Yaskawa INFORM job: X2_99(90,0)_HARDOX.JBI

/JOB
//NAME X2_99(90,0)_HARDOX
///FOLDERNAME X2
//POS
///NPOS 447,447,443,13,0,0
///TOOL 0
///POSTYPE PULSE
///PULSE
C00000=2000,-99612,-82443,0,53832,0
C00001=-166393,-132062,-92618,58483,55149,81008
C00002=-157482,-99612,-82443,50725,53832,-76817
C00003=-152781,-96239,-78741,49340,50884,-75750
C00004=-150954,-94792,-77210,48744,49760,-75306
C00005=-150957,-94045,-75225,49281,49201,-75681
C00006=-151067,-94769,-77060,48840,49767,-75375
C00007=-148896,-96259,-77631,48213,48319,-74911
C00008=-154925,-106114,-81211,52368,49780,-77962
C00009=-154976,-104737,-78409,53070,49177,-78455
C00010=-153765,-101609,-77307,52041,49068,-77683
C00011=-154727,-103781,-80113,51957,49998,-77663
C00012=-157482,-99612,-82443,50725,53832,-76817
C00013=-126812,-81448,-90767,9472,77282,-14340
C00014=-120783,-85892,-98127,-47,82159,60
C00015=-120791,-78998,-92147,-45,82022,58
C00016=-120812,-59041,-81112,-38,85486,50
C00017=-120812,-59638,-79752,-38,84341,50
C00018=-120812,-59041,-81112,-38,85486,50
C00019=-120792,-70899,-87175,-45,83124,57
C00020=-120810,-72484,-85548,-40,81307,51
C00021=-120817,-76009,-87202,-37,80512,50
C00022=-120816,-72927,-85752,-37,81205,50
C00023=-120792,-71723,-87920,-45,83159,57
C00024=-120783,-85892,-98127,-47,82159,60
C00025=-120841,-86418,-98444,-30,82084,41
C00026=-120867,-62955,-84955,-21,85839,32
C00027=-120862,-57449,-80347,-23,85833,34
C00028=-120862,-58065,-78999,-24,84687,34
C00029=-120862,-57449,-80347,-23,85833,34
C00030=-120848,-76846,-90076,-28,81853,39
C00031=-120700,-77430,-87681,-72,80079,89
C00032=-120707,-73445,-85814,-70,80978,86
C00033=-120700,-77430,-87681,-72,80079,89
C00034=-120841,-86418,-98444,-30,82084,41
C00035=-120877,-85820,-98106,-19,82183,30
C00036=-120894,-60284,-82721,-14,85837,23
C00037=-120891,-57831,-80469,-15,85712,24
C00038=-120891,-58439,-79117,-15,84567,25
C00039=-120891,-57831,-80469,-15,85712,24
C00040=-120882,-76306,-89742,-18,81925,28
C00041=-120632,-76849,-87581,-92,80316,111
C00042=-120641,-72870,-85708,-89,81208,107
C00043=-120899,-105607,-111704,-13,80383,24
C00044=-120899,-105607,-111704,-13,80383,24
C00045=-120329,-64675,-84682,-181,84785,205
C00046=-120337,-61857,-81845,-179,84488,203
C00047=-120337,-62228,-80870,-179,83698,204
C00048=-120337,-61849,-81865,-179,84506,203
C00049=-120308,-72964,-87409,-188,82206,216
C00050=-112365,-66887,-81837,-2540,82030,2815
C00051=-112466,-65041,-80903,-2509,82400,2777
C00052=-112291,-68228,-82506,-2565,81755,2847
C00053=-88690,-37051,-64863,-22386,100281,29037
C00054=-90338,-32373,-60570,-22143,99643,28585
C00055=-86677,-30127,-56933,-28301,101078,28609
C00056=-87262,-30704,-57322,-28229,100840,28451
C00057=-86036,-30845,-57417,-28365,101220,28810
C00058=-80749,-50154,-73696,-28906,103010,30322
C00059=-106026,-92840,-102541,-4408,81700,4909
C00060=-104933,-21068,-63327,-14588,98299,15445
C00061=-118026,-7058,-59426,2478,121298,42537
C00062=-119206,-9959,-57512,2402,118662,42076
C00063=-119679,-11008,-56668,2374,117617,41892
C00064=-119678,-12040,-55711,2348,116499,41868
C00065=-119679,-11008,-56668,2374,117617,41892
C00066=-117888,-11929,-55575,2351,116426,42475
C00067=-118578,-11982,-55616,2350,116441,42241
C00068=-117888,-11929,-55575,2351,116426,42475
C00069=-116239,-8118,-58416,2447,120087,43116
C00070=-117941,-7017,-59404,2478,121303,42566
C00071=-119121,-9922,-57492,2402,118667,42105
C00072=-119594,-10972,-56650,2375,117622,41921
C00073=-119593,-12004,-55694,2348,116504,41897
C00074=-119594,-10972,-56650,2375,117622,41921
C00075=-117972,-11968,-55595,2351,116420,42446
C00076=-118663,-12020,-55635,2349,116436,42212
C00077=-117972,-11968,-55595,2351,116420,42446
C00078=-116323,-8162,-58441,2447,120082,43087
C00079=-118213,-4464,-57342,2479,121353,42475
C00080=-119375,-7335,-55445,2404,118742,42020
C00081=-119840,-8375,-54609,2376,117706,41839
C00082=-119839,-9401,-53662,2350,116597,41815
C00083=-119840,-8375,-54609,2376,117706,41839
C00084=-117787,-9255,-53494,2353,116516,42511
C00085=-118466,-9310,-53537,2352,116532,42281
C00086=-117787,-9255,-53494,2353,116516,42511
C00087=-113921,-56504,-90793,-659,90254,43086
C00088=-172997,-84117,-74043,29270,60841,12459
C00089=-182497,-62439,-47217,33561,35566,5540
C00090=-177866,51889,12751,25241,78726,20035
C00091=-177567,56483,20827,25353,76270,19609
C00092=-176984,60218,26227,25284,74822,19505
C00093=-176718,63716,30232,25261,74138,19453
C00094=-180313,74951,43422,33206,78652,20175
C00095=-180313,74899,44483,33273,78081,20005
C00096=-179620,70269,37422,31209,78046,20027
C00097=-177875,51523,13769,25307,77989,19872
C00098=-167005,53799,14731,23971,77323,24144
C00099=-166588,57735,22127,23390,74500,23603
C00100=-166048,58751,23437,20984,72747,23092
C00101=-165731,62483,27692,20928,72014,23074
C00102=-170479,73702,41207,33101,77375,24075
C00103=-170176,75335,43164,33053,76951,24069
C00104=-170176,75225,45395,33224,75746,23705
C00105=-170176,75310,43480,33077,76778,24016
C00106=-166977,49436,12685,24253,74137,23502
C00107=-182364,4853,-37106,25072,86261,16971
C00108=-152303,-102933,-107906,-365,71882,21471
C00109=-90355,-23252,-64713,-31290,93997,-15055
C00110=-138081,35844,8180,-39695,66399,-31141
C00111=-138669,40694,16134,-40133,64268,-30541
C00112=-138897,42750,19469,-40345,63394,-30283
C00113=-139039,48061,25142,-40529,62744,-30077
C00114=-139353,43961,18205,-39728,64276,-30868
C00115=-137559,60892,31006,-35555,70429,-31778
C00116=-137559,60794,32915,-35805,69424,-31435
C00117=-137731,58187,28052,-35412,70711,-31945
C00118=-138069,35590,9192,-39905,65818,-30900
C00119=-133067,14417,-5479,-38193,49171,-52584
C00120=-129431,19961,2498,-38515,39991,-63248
C00121=-130261,24926,10174,-39520,37911,-62617
C00122=-130583,27008,13377,-40001,37063,-62330
C00123=-131019,32231,18551,-40077,36476,-62276
C00124=-130460,44452,16810,-29784,55193,-70193
C00125=-130349,47098,21751,-30441,53767,-69689
C00126=-130349,47115,24243,-31014,52449,-69252
C00127=-130073,43731,18555,-30519,54073,-69657
C00128=-124769,26347,15261,-56693,39526,-56291
C00129=-125951,31366,21174,-57124,38215,-56008
C00130=-125990,33793,23574,-57346,38066,-55879
C00131=-123661,25065,17775,-59577,38998,-54642
C00132=-126326,41414,28236,-49768,42989,-60672
C00133=-126284,55009,36720,-51578,51165,-54455
C00134=-126583,51433,35812,-56160,48613,-52922
C00135=-130309,48205,31707,-53943,60165,-33503
C00136=-132420,66802,42698,-49866,69800,-28677
C00137=-133401,41961,21720,-50712,64405,-25968
C00138=-132439,36745,15005,-50531,65875,-26297
C00139=-90355,-25240,-62492,-31182,91940,-14489
C00140=-126181,-67140,-93758,-13250,84858,5822
C00141=-152303,-102933,-107906,-365,71882,21471
C00142=-151021,-50166,-89002,-846,87371,21807
C00143=-182364,4853,-37106,25072,86261,16971
C00144=-184325,60344,23585,34019,76352,15866
C00145=-184220,82357,46305,33005,82595,16795
C00146=-183957,81689,47427,34502,79595,16153
C00147=-184996,71033,34569,34595,82030,16501
C00148=-182797,88211,55548,32842,79786,16530
C00149=-166812,83754,46609,21700,79823,22205
C00150=-169419,57666,21738,28270,70846,20124
C00151=-169758,52135,14437,28170,72420,20393
C00152=-182364,4853,-37106,25072,86261,16971
C00153=-152303,-102933,-107906,-365,71882,21471
C00154=-121799,-34443,-59064,-1710,93632,36707
C00155=-118945,163,-15392,-1659,93503,40633
C00156=-120696,28796,14633,-1549,89703,40093
C00157=-120697,41895,29242,-1556,93940,40040
C00158=-120696,45752,33571,-1566,96736,40005
C00159=-120665,21626,9251,-1581,100352,39971
C00160=-120660,1326,-9108,-1544,99287,41805
C00161=-120641,1282,-9371,-1543,99426,41811
C00162=-120163,-1908,-13337,-1516,100237,41964
C00163=-118931,-1420,-16721,-1449,102592,42361
C00164=-118945,163,-15392,-1659,93503,40633
C00165=-120171,930,-10959,-1582,91145,40250
C00166=-120660,1326,-9108,-1553,90200,40098
C00167=-120694,25865,13192,-1550,89085,40100
C00168=-120696,29026,16285,-1550,88805,40104
C00169=-120258,23290,9189,-1576,90234,40233
C00170=-119165,22386,4533,-1644,92655,40570
C00171=-119181,24192,6266,-1459,101602,42286
C00172=-120260,23811,9690,-1517,99280,41943
C00173=-120693,23749,11149,-1541,98342,41806
C00174=-120660,1326,-9108,-1544,99287,41805
C00175=-120174,1432,-10536,-1517,100229,41961
C00176=-118965,1918,-13913,-1451,102579,42349
C00177=-119164,21752,3941,-1459,101779,42290
C00178=-120255,21351,7351,-1518,99456,41942
C00179=-120694,21281,8802,-1542,98518,41803
C00180=-120641,1282,-9371,-1543,99426,41811
C00181=-120163,-1908,-13337,-1516,100237,41964
C00182=-118931,-1420,-16721,-1449,102592,42361
C00183=-109578,15420,-7310,-28367,110236,-41857
C00184=-109763,14188,-4345,-27924,107995,-41350
C00185=-110193,13805,-2890,-27787,106881,-41239
C00186=-131022,13378,-3260,-29129,99839,-47636
C00187=-122106,10683,8881,-53521,92538,-44133
C00188=-120623,10562,7326,-53535,93941,-44154
C00189=-119164,10594,3761,-53715,96134,-44669
C00190=-115308,-32515,-29810,-53374,97452,-43308
C00191=-160324,-56725,-62447,4686,86573,-10750
C00192=-150232,17988,-5017,26557,112251,35280
C00193=-142954,11495,-10959,27504,110227,37702
C00194=-142768,10690,-7556,27067,107926,37200
C00195=-143003,11007,-5424,26849,106972,36875
C00196=-137789,7639,-8393,27391,105376,38540
C00197=-140743,9596,5422,48538,102657,38323
C00198=-145934,20226,29397,62426,105383,26201
C00199=-142397,10029,6905,51885,103476,38119
C00200=-144627,12481,5478,52145,106089,38424
C00201=-150232,17988,-5017,26557,112251,35280
C00202=-160324,-56725,-62447,4686,86573,-10750
C00203=-146496,-53907,-57071,50358,82742,77471
C00204=-142086,-46087,-49611,49702,79955,78251
C00205=-140910,-47839,-49478,49629,78666,78171
C00206=-141016,-46873,-48908,49627,78820,78198
C00207=-140042,-41059,-45363,49344,78825,78701
C00208=-141209,-66264,-43604,72924,53654,56912
C00209=-144414,-64476,-42796,72863,55989,56716
C00210=-142865,-68044,-45540,72856,54877,56844
C00211=-146705,-71229,-49721,72532,57818,56833
C00212=-150615,-73008,-67005,51145,82624,75252
C00213=-84213,-62636,-84550,-16381,94117,81885
C00214=-95245,-30826,-59151,-14149,92862,78402
C00215=-96701,-43295,-61552,-15492,82772,78870
C00216=-98227,-44091,-62190,-15063,82479,78389
C00217=-94037,-41035,-61513,-16198,84364,79567
C00218=-63521,1839,6360,-71273,102323,80160
C00219=-65232,-1066,5117,-71288,100899,80280
C00220=-65232,-364,7293,-71071,100558,80717
C00221=-61873,133,7709,-70638,102845,81131
C00222=-97631,-84017,-82277,-6042,71977,80454
C00223=-97631,-84017,-82277,-6042,71977,13540
C00224=-100992,-100869,-74320,-15072,37892,15545
C00225=-103157,-95187,-70426,-13089,38023,14317
C00226=-103157,-92961,-65713,-13621,36312,14617
C00227=-97699,-120955,-80408,-20799,32327,18909
C00228=2000,-45096,-51939,0,82773,0
C00229=2000,-45096,-51939,0,82773,0
C00230=2000,-45096,-51939,0,82773,0
C00231=2000,-45096,-51939,0,82773,0
C00232=2000,-45096,-51939,0,82773,0
C00233=-70410,-104162,-83449,-55661,60383,81011
C00234=-84923,-92751,-76765,-50721,53081,76684
C00235=-86734,-91468,-75289,-50215,51915,76295
C00236=-86736,-90744,-73307,-50726,51361,76670
C00237=-86623,-91438,-75136,-50303,51925,76361
C00238=-88689,-93063,-75778,-49797,50498,75974
C00239=-86623,-91438,-75136,-50303,51925,76361
C00240=-82499,-102310,-79219,-53526,52313,78845
C00241=-82460,-100986,-76424,-54186,51705,79335
C00242=-83746,-97994,-75341,-53258,51491,78599
C00243=-82460,-100986,-76424,-54186,51705,79335
C00244=-83820,-89231,-90898,-31984,73153,45470
C00245=-103333,-81093,-95821,-5106,83352,5547
C00246=-105734,-58391,-81894,-4383,86302,4664
C00247=-106051,-55558,-79074,-4290,86007,4572
C00248=-106052,-56155,-77720,-4294,84870,4611
C00249=-106051,-55558,-79074,-4290,86007,4572
C00250=-104417,-72181,-87594,-4790,82806,5215
C00251=-104401,-72744,-85473,-4810,81218,5281
C00252=-104801,-68935,-83629,-4684,82015,5119
C00253=-104401,-72744,-85473,-4810,81218,5281
C00254=-103333,-81093,-95821,-5106,83352,5547
C00255=-121034,-86160,-98106,184,81635,-191
C00256=-120937,-60313,-84022,154,86250,-153
C00257=-120931,-57182,-80055,152,85416,-152
C00258=-120931,-57770,-78693,152,84276,-154
C00259=-120931,-57182,-80055,152,85416,-152
C00260=-120995,-76536,-89732,172,81427,-178
C00261=-121142,-77068,-87314,217,79666,-229
C00262=-121124,-73096,-85459,211,80565,-222
C00263=-121142,-77068,-87314,217,79666,-229
C00264=-121096,-115670,-111851,205,74930,-222
C00265=-121096,-115670,-111851,205,74930,-222
C00266=-111920,-77360,-89293,-2569,80863,2809
C00267=-113418,-69208,-82911,-2118,81083,2310
C00268=-113298,-70113,-82134,-2157,80142,2365
C00269=-113298,-69851,-83365,-2151,81033,2349
C00270=-112830,-79068,-87705,-2304,78982,2541
C00271=-118405,-74923,-83336,-614,78322,682
C00272=-118432,-73250,-82545,-605,78695,671
C00273=-118359,-77891,-84712,-629,77644,701
C00274=-147649,-49700,-70143,21952,96038,-28312
C00275=-144092,-44169,-65180,21423,94945,-27268
C00276=-143301,-44665,-65479,21298,94683,-27039
C00277=-145130,-43494,-64769,21581,95292,-27566
C00278=-153783,-86392,-93366,22522,93398,-30972
C00279=-150910,-93017,-97560,17688,85250,-21630
C00280=-120908,-62091,-84868,144,85857,-144
C00281=-120903,-58004,-80414,143,85215,-144
C00282=-120903,-58580,-79044,143,84076,-145
C00283=-120903,-58004,-80414,143,85215,-144
C00284=-120961,-76486,-89626,161,81387,-167
C00285=-121210,-76970,-87437,238,79792,-251
C00286=-121190,-72994,-85579,231,80691,-243
C00287=-121210,-76970,-87437,238,79792,-251
C00288=-120997,-86105,-97999,172,81597,-178
C00289=-122173,-44832,-80249,-1138,103105,-21360
C00290=-123342,-6609,-59067,-2432,120936,-42504
C00291=-122164,-9458,-57119,-2365,118305,-42047
C00292=-121693,-10486,-56262,-2341,117263,-41864
C00293=-121692,-11496,-55292,-2315,116147,-41841
C00294=-121693,-10486,-56262,-2341,117263,-41864
C00295=-123477,-11388,-55156,-2308,116075,-42444
C00296=-122789,-11440,-55197,-2311,116090,-42211
C00297=-123477,-11388,-55156,-2308,116075,-42444
C00298=-125124,-7649,-58044,-2392,119728,-43080
C00299=-123427,-6569,-59045,-2432,120941,-42533
C00300=-122249,-10161,-56477,-2346,117547,-42058
C00301=-121777,-10451,-56245,-2341,117268,-41893
C00302=-121777,-11461,-55275,-2315,116153,-41870
C00303=-121777,-10451,-56245,-2341,117268,-41893
C00304=-123393,-11428,-55177,-2309,116069,-42415
C00305=-122704,-11478,-55216,-2311,116085,-42182
C00306=-123393,-11428,-55177,-2309,116069,-42415
C00307=-123141,-2998,-56146,-2434,120999,-42438
C00308=-121991,-6366,-54527,-2366,118305,-41988
C00309=-121527,-6824,-53376,-2344,117373,-41811
C00310=-121527,-7826,-52419,-2319,116269,-41787
C00311=-121527,-6824,-53376,-2344,117373,-41811
C00312=-123560,-7684,-52253,-2311,116189,-42474
C00313=-122887,-7737,-52295,-2313,116204,-42247
C00314=-123560,-7684,-52253,-2311,116189,-42474
C00315=-125171,-3981,-55094,-2393,119797,-43097
C00316=-101327,-45531,-60072,-2075,102128,-34667
C00317=-89266,4396,-33928,-11465,93507,-29927
C00318=-79229,40490,546,-19170,75952,-25029
C00319=-79192,44826,8093,-19384,73673,-24644
C00320=-79178,46660,11239,-19482,72737,-24484
C00321=-79430,50869,15806,-19440,72068,-24459
C00322=-81284,59295,20499,-15163,78789,-25581
C00323=-81374,60489,21858,-15140,78557,-25582
C00324=-81374,60030,23342,-15197,77446,-25442
C00325=-81374,60441,21998,-15146,78450,-25567
C00326=-79222,40075,1538,-19236,75173,-24900
C00327=-94467,40678,813,-12417,73109,-29814
C00328=-94083,44902,8245,-12754,70817,-29441
C00329=-93934,46692,11343,-12898,69876,-29287
C00330=-93910,50579,15562,-12974,69302,-29211
C00331=-93927,66497,27908,-12345,79633,-30207
C00332=-93899,67606,29206,-12360,79415,-30175
C00333=-93899,67330,30165,-12386,78699,-30102
C00334=-93899,67593,29245,-12361,79385,-30171
C00335=-94477,40302,1770,-12461,72343,-29738
C00336=-89266,4396,-33928,-11465,93507,-29927
C00337=-101327,-45531,-60072,-2075,102128,-34667
C00338=-154347,-58865,-59313,31959,84488,20300
C00339=-132804,-7309,-34611,38234,83249,26564
C00340=-122368,37716,10148,50470,78338,25854
C00341=-122011,44734,21095,50873,76111,24806
C00342=-122399,46275,23078,51041,76048,24565
C00343=-121689,49763,26849,50970,75314,24530
C00344=-120622,58400,25662,45422,83740,28939
C00345=-120341,59602,27023,45371,83444,28935
C00346=-120341,59440,28250,45426,82846,28662
C00347=-120341,59624,26889,45365,83513,28966
C00348=-125132,37819,11526,51275,79326,24970
C00349=-124576,6255,-12780,47438,56902,47453
C00350=-122250,19334,1935,46182,44641,59320
C00351=-122250,19334,1935,46182,44641,59320
C00352=-120782,25934,12333,47564,41782,58376
C00353=-120333,29516,15843,47539,41325,58369
C00354=-116027,40200,8001,22624,59086,67088
C00355=-115770,42313,10216,22534,58761,67121
C00356=-115770,42134,11170,22690,58133,66983
C00357=-116328,39236,6565,22717,59528,67061
C00358=-134725,35683,25951,66201,49933,50817
C00359=-134127,37360,27871,66271,49401,50755
C00360=-134767,35094,27603,67235,49407,50088
C00361=-133752,44861,29735,56261,55408,56901
C00362=-130842,31560,20725,61115,49473,53899
C00363=-126547,58238,34123,55061,83310,26481
C00364=-128263,40961,20002,56228,76218,21701
C00365=-128172,35801,14205,55931,76570,22030
C00366=-132804,-7309,-34611,38234,83249,26564
C00367=-154347,-58865,-59313,31959,84488,20300
C00368=-101327,-45531,-60072,-2075,102128,-34667
C00369=-89266,4396,-33928,-11465,93507,-29927
C00370=-72391,40299,1753,-27854,73409,-20952
C00371=-72736,45425,8735,-27946,71826,-20687
C00372=-74859,57115,18605,-23013,76545,-21887
C00373=-89811,68744,24857,-14650,79648,-27077
C00374=-89486,63951,21050,-15706,77371,-26858
C00375=-88154,41926,3429,-20512,68875,-25737
C00376=-87331,-25296,-55522,-7683,87670,-26764
C00377=-122403,540,-15029,1679,93098,-40614
C00378=-120549,50049,35393,1611,98655,-39918
C00379=-120549,50860,39291,1601,96673,-39943
C00380=-120548,50863,39319,1606,97508,-39933
C00381=-120592,23246,10920,1617,100389,-39913
C00382=-120666,1773,-8688,1564,98883,-41779
C00383=-120644,766,-9415,1564,98810,-41771
C00384=-121185,-971,-12517,1537,99838,-41946
C00385=-122412,-533,-15942,1476,102193,-42339
C00386=-122403,540,-15029,1679,93098,-40614
C00387=-121179,1356,-10556,1597,90741,-40233
C00388=-120574,1774,-8687,1557,89793,-40041
C00389=-120532,26429,13697,1554,88684,-40039
C00390=-121099,23723,9564,1591,89850,-40218
C00391=-122190,22771,4863,1663,92275,-40553
C00392=-122175,24579,6594,1485,101224,-42269
C00393=-121098,24245,10065,1538,98897,-41927
C00394=-120630,24202,11544,1561,97957,-41779
C00395=-120666,1773,-8688,1564,98883,-41779
C00396=-121177,1858,-10134,1538,99825,-41943
C00397=-122384,2295,-13553,1478,102176,-42330
C00398=-122189,22661,4761,1485,101367,-42272
C00399=-121101,22312,8220,1538,99039,-41927
C00400=-120664,22262,9692,1560,98100,-41789
C00401=-120644,766,-9415,1564,98810,-41771
C00402=-121185,-971,-12517,1537,99838,-41946
C00403=-122412,-533,-15942,1476,102193,-42339
C00404=-131781,15460,-7279,28376,109886,41795
C00405=-131592,14275,-4268,27940,107640,41290
C00406=-131503,14118,-2773,27783,106722,41093
C00407=-110365,13875,-2999,29065,99587,47581
C00408=-120145,11200,9350,53476,92778,43812
C00409=-120732,10849,7590,53521,93669,44023
C00410=-122191,10834,3980,53696,95864,44539
C00411=-128646,-26020,-30624,53883,101032,13133
C00412=-66557,-34885,-48546,-20214,102394,-2504
C00413=-79484,36547,13079,-24373,114005,-30975
C00414=-85904,26694,3247,-25718,112997,-33343
C00415=-86041,25965,6661,-25253,110710,-32858
C00416=-86402,26110,8646,-25107,109560,-32737
C00417=-90488,21267,4070,-25796,108613,-34139
C00418=-88154,25384,22913,-49666,108029,-34753
C00419=-86352,23519,22887,-52150,107314,-32505
C00420=-84237,28413,32993,-57339,108017,-31709
C00421=-87086,25419,21214,-49770,109322,-34894
C00422=-85922,26350,18486,-50250,111381,-35429
C00423=-81578,31234,5255,-15438,110633,-30982
C00424=-71416,-31459,-49219,-37385,106309,-54903
C00425=-79334,-27512,-40554,-52438,93314,-75230
C00426=-81671,-29746,-39165,-52092,90747,-74997
C00427=-82927,-31826,-39398,-51944,89460,-74930
C00428=-82828,-30765,-38686,-51956,89581,-74947
C00429=-84254,-26168,-35546,-51810,89054,-75403
C00430=-79369,-49621,-34755,-72713,68891,-55712
C00431=-83639,-30110,-37749,-52241,83019,-70160
C00432=-77493,-50941,-36554,-72626,70323,-55695
C00433=-74018,-52299,-39928,-72336,73171,-55924
C00434=-60945,-55409,-65093,-53734,104166,-71681
C00435=-60945,-55409,-65093,-53734,104166,-71681
C00436=-127789,-76367,-82464,-10340,71927,-66680
C00437=-126395,-68335,-70990,-10768,62738,-65273
C00438=-128368,-67800,-70596,-9819,62518,-66000
C00439=-129736,-90807,-85563,-9383,59779,-66288
C00440=-134440,-102926,-90239,1517,55386,-10396
C00441=-137693,-99872,-71253,8781,33093,-13294
C00442=-140882,-99069,-62349,23538,21711,-19417
C00443=-140882,-96084,-57211,25293,20222,-20256
C00444=-141874,-99800,-58459,28296,19507,-21772
C00445=-122092,-114409,-88723,8345,70481,-11232
C00446=2000,-48025,-60869,0,102856,0
BC00000=0,666204,302418
BC00001=33147,674408,66891
BC00002=34043,674630,60526
BC00003=34043,674630,60526
BC00004=34043,674630,60526
BC00005=34043,674630,60526
BC00006=34043,674630,60526
BC00007=34043,674630,60526
BC00008=34043,674630,60526
BC00009=34043,674630,60526
BC00010=34043,674630,60526
BC00011=34043,674630,60526
BC00012=34043,674630,60526
BC00013=15644,667481,91364
BC00014=12814,672902,59330
BC00015=12814,672902,59330
BC00016=12814,672902,59330
BC00017=12814,672902,59330
BC00018=12814,672902,59330
BC00019=12814,672902,59330
BC00020=12814,672902,59330
BC00021=12814,672902,59330
BC00022=12814,672902,59330
BC00023=12814,672902,59330
BC00024=12814,672902,59330
BC00025=70623,673655,58742
BC00026=70623,673655,58742
BC00027=70623,673655,58742
BC00028=70623,673655,58742
BC00029=70623,673655,58742
BC00030=70623,673655,58742
BC00031=70623,673655,58742
BC00032=70623,673655,58742
BC00033=70623,673655,58742
BC00034=70623,673655,58742
BC00035=129248,673621,59299
BC00036=129248,673621,59299
BC00037=129248,673621,59299
BC00038=129248,673621,59299
BC00039=129248,673621,59299
BC00040=129248,673621,59299
BC00041=129248,673621,59299
BC00042=129248,673621,59299
BC00043=129248,669709,59299
BC00044=389488,669709,59299
BC00045=389488,669709,59299
BC00046=389488,669709,59299
BC00047=389488,669709,59299
BC00048=389488,669709,59299
BC00049=389488,669709,59299
BC00050=389488,669709,59299
BC00051=389488,669709,59299
BC00052=389488,669709,59299
BC00053=389488,669709,59299
BC00054=389488,669709,59299
BC00055=389488,669709,59299
BC00056=389488,669709,59299
BC00057=389488,669709,59299
BC00058=389488,669709,59299
BC00059=129248,671899,59299
BC00060=129248,671899,59299
BC00061=131979,699465,58241
BC00062=131979,699465,58241
BC00063=131979,699465,58241
BC00064=131979,699465,58241
BC00065=131979,699465,58241
BC00066=131979,699465,58241
BC00067=131979,699465,58241
BC00068=131979,699465,58241
BC00069=131979,699465,58241
BC00070=132002,746034,57968
BC00071=132002,746034,57968
BC00072=132002,746034,57968
BC00073=132002,746034,57968
BC00074=132002,746034,57968
BC00075=132002,746034,57968
BC00076=132002,746034,57968
BC00077=132002,746034,57968
BC00078=132002,746034,57968
BC00079=131294,789553,57813
BC00080=131294,789553,57813
BC00081=131294,789553,57813
BC00082=131294,789553,57813
BC00083=131294,789553,57813
BC00084=131294,789553,57813
BC00085=131294,789553,57813
BC00086=131294,789553,57813
BC00087=131294,789553,57813
BC00088=183654,789553,192797
BC00089=205319,789553,241609
BC00090=192952,789553,63191
BC00091=192952,789553,63191
BC00092=192952,789553,63191
BC00093=192952,789553,63191
BC00094=192952,789553,63191
BC00095=192952,789553,63191
BC00096=192952,789553,63191
BC00097=192952,789553,63191
BC00098=197720,789553,63337
BC00099=197720,789553,63337
BC00100=197720,789553,63337
BC00101=197720,789553,63337
BC00102=197719,789553,63336
BC00103=197719,789553,63336
BC00104=197719,789553,63336
BC00105=197719,789553,63336
BC00106=197720,789553,63337
BC00107=190214,789553,90491
BC00108=160526,789553,32122
BC00109=129825,789553,81519
BC00110=178627,789553,88525
BC00111=178627,789553,88525
BC00112=178627,789553,88525
BC00113=178627,789553,88521
BC00114=178627,789553,88521
BC00115=178627,786924,70712
BC00116=178627,786924,70712
BC00117=178627,786924,70712
BC00118=178627,789553,88525
BC00119=173223,789553,85007
BC00120=170379,789553,83156
BC00121=170379,789553,83156
BC00122=170379,789553,83156
BC00123=170379,789553,83155
BC00124=170379,789553,83155
BC00125=170379,789553,83155
BC00126=170379,789553,83155
BC00127=170379,789553,83155
BC00128=170693,789553,81519
BC00129=170693,789553,81519
BC00130=170693,789553,81519
BC00131=170693,789553,81519
BC00132=170693,789553,81519
BC00133=170693,780224,54167
BC00134=170693,780224,54167
BC00135=170693,789366,80970
BC00136=170693,779782,47084
BC00137=170693,789553,81519
BC00138=170693,789553,81519
BC00139=129825,789553,81519
BC00140=147580,789553,52951
BC00141=160526,789553,32122
BC00142=160526,789553,32122
BC00143=190214,789553,90491
BC00144=205319,789553,32122
BC00145=205319,789553,32121
BC00146=205319,789553,32122
BC00147=205319,789553,32122
BC00148=205319,789553,32121
BC00149=205319,789553,32122
BC00150=205319,789553,32122
BC00151=205319,789553,32122
BC00152=190214,789553,90491
BC00153=160526,789553,32122
BC00154=125912,765497,191733
BC00155=143425,748886,281271
BC00156=143425,748886,281271
BC00157=143425,748886,281271
BC00158=143425,748886,281271
BC00159=143425,748886,281271
BC00160=143559,719962,281608
BC00161=143735,675447,281889
BC00162=143735,675447,281889
BC00163=143735,675447,281889
BC00164=143425,748886,281271
BC00165=143425,748886,281271
BC00166=143425,748886,281271
BC00167=143425,748886,281271
BC00168=143425,748886,281271
BC00169=143425,748886,281271
BC00170=143425,748886,281271
BC00171=143559,719962,281608
BC00172=143559,719962,281608
BC00173=143559,719962,281608
BC00174=143559,719962,281608
BC00175=143559,719962,281608
BC00176=143559,719962,281608
BC00177=143735,675447,281889
BC00178=143735,675447,281889
BC00179=143735,675447,281889
BC00180=143735,675447,281889
BC00181=143735,675447,281889
BC00182=143735,675447,281889
BC00183=146695,666220,221883
BC00184=146695,666220,221883
BC00185=146695,666220,221883
BC00186=146695,666220,221883
BC00187=146695,666220,221881
BC00188=146695,666220,221883
BC00189=146695,666220,221883
BC00190=146695,666220,221883
BC00191=15,666220,224435
BC00192=15,666220,224435
BC00193=15,666220,224435
BC00194=15,666220,224435
BC00195=15,666220,224435
BC00196=15,666220,224435
BC00197=15,666220,224435
BC00198=15,666220,224435
BC00199=15,666220,224435
BC00200=15,666220,224435
BC00201=15,666220,224435
BC00202=15,666220,224435
BC00203=16,666221,121466
BC00204=15,666220,121470
BC00205=15,666220,121470
BC00206=15,666220,121470
BC00207=15,666220,121470
BC00208=15,666220,121470
BC00209=15,666220,121470
BC00210=15,666220,121470
BC00211=15,666220,121470
BC00212=15,666220,121470
BC00213=383087,666220,121470
BC00214=383087,666220,121470
BC00215=383087,666220,121470
BC00216=383087,666220,121470
BC00217=383087,666220,121470
BC00218=383087,666220,121470
BC00219=383087,666220,121470
BC00220=383087,666220,121470
BC00221=383087,666220,121470
BC00222=383087,666220,121470
BC00223=383087,666220,121470
BC00224=383087,666220,121470
BC00225=383087,666220,121470
BC00226=383087,666220,121470
BC00227=383087,666220,121470
BC00228=15,666220,1075229
BC00229=15,666220,1075229
BC00230=15,666220,1075229
BC00231=15,666220,1075229
BC00232=15,666220,1075229
BC00233=398174,675740,57967
BC00234=398174,675740,57967
BC00235=398174,675740,57967
BC00236=398174,675740,57967
BC00237=398174,675740,57967
BC00238=398174,675740,57967
BC00239=398174,675740,57967
BC00240=398174,675740,57967
BC00241=398174,675740,57967
BC00242=398174,675740,57967
BC00243=398174,675740,57967
BC00244=398174,674932,57390
BC00245=398174,674023,56741
BC00246=398174,674023,56741
BC00247=398174,674023,56741
BC00248=398174,674023,56741
BC00249=398174,674023,56741
BC00250=398174,674023,56741
BC00251=398174,674023,56741
BC00252=398174,674023,56741
BC00253=398174,674023,56741
BC00254=398174,674023,56741
BC00255=366924,674754,56144
BC00256=366924,674754,56144
BC00257=366924,674754,56144
BC00258=366924,674754,56144
BC00259=366924,674754,56144
BC00260=366924,674754,56144
BC00261=366924,674754,56144
BC00262=366924,674754,56144
BC00263=366924,674754,56144
BC00264=366924,674754,56144
BC00265=30712,674754,56144
BC00266=30712,674754,68643
BC00267=30712,674754,68643
BC00268=30712,674754,68643
BC00269=30712,674754,68643
BC00270=30712,674754,68643
BC00271=30712,674754,68643
BC00272=30712,674754,68643
BC00273=30712,674754,68643
BC00274=30712,674754,68643
BC00275=30712,674754,68643
BC00276=30712,674754,68643
BC00277=30712,674754,68643
BC00278=30712,674754,68643
BC00279=339116,680642,91140
BC00280=308298,674696,56672
BC00281=308298,674696,56672
BC00282=308298,674696,56672
BC00283=308298,674696,56672
BC00284=308298,674696,56672
BC00285=308298,674696,56672
BC00286=308298,674696,56672
BC00287=308298,674696,56672
BC00288=308298,674696,56672
BC00289=306928,687618,56444
BC00290=305557,700540,56217
BC00291=305557,700540,56217
BC00292=305557,700540,56217
BC00293=305557,700540,56217
BC00294=305557,700540,56217
BC00295=305557,700540,56217
BC00296=305557,700540,56217
BC00297=305557,700540,56217
BC00298=305557,700540,56217
BC00299=305514,747109,57030
BC00300=305514,747109,57030
BC00301=305514,747109,57030
BC00302=305514,747109,57030
BC00303=305514,747109,57030
BC00304=305514,747109,57030
BC00305=305514,747109,57030
BC00306=305514,747109,57030
BC00307=306202,789553,57955
BC00308=306202,789553,57955
BC00309=306202,789553,57955
BC00310=306202,789553,57955
BC00311=306202,789553,57955
BC00312=306202,789553,57955
BC00313=306202,789553,57955
BC00314=306202,789553,57955
BC00315=306202,789553,57955
BC00316=306202,789553,221991
BC00317=298504,779638,136331
BC00318=292117,771411,65252
BC00319=292117,771411,65252
BC00320=292117,771411,65252
BC00321=292117,771411,65252
BC00322=292117,771411,65252
BC00323=292117,771411,65252
BC00324=292117,771411,65252
BC00325=292117,771411,65252
BC00326=292117,771411,65252
BC00327=297138,774664,65917
BC00328=297138,774664,65917
BC00329=297138,774664,65917
BC00330=297137,774662,65916
BC00331=297137,774662,65916
BC00332=297137,774662,65916
BC00333=297137,774662,65916
BC00334=297137,774662,65916
BC00335=297138,774664,65917
BC00336=298504,779638,136331
BC00337=306202,789553,221991
BC00338=306202,789553,221991
BC00339=301081,789553,147340
BC00340=309933,789553,80201
BC00341=309933,789553,80201
BC00342=309933,789553,80201
BC00343=309933,789553,80200
BC00344=309933,789553,44577
BC00345=309933,789553,44577
BC00346=309933,789553,44577
BC00347=309933,789553,44577
BC00348=309933,789553,80201
BC00349=297228,789553,85661
BC00350=297336,789553,84334
BC00351=297336,789553,84334
BC00352=297336,789553,84334
BC00353=297336,789553,84334
BC00354=297336,789553,53509
BC00355=297336,789553,53509
BC00356=297336,789553,53509
BC00357=297336,789553,53509
BC00358=326204,789553,82063
BC00359=326204,789553,82063
BC00360=326204,789553,82063
BC00361=326204,789553,82063
BC00362=326204,789553,82063
BC00363=326152,789553,55059
BC00364=326201,789553,82063
BC00365=326204,789553,82063
BC00366=301081,789553,147340
BC00367=306202,789553,221991
BC00368=306202,789553,221991
BC00369=298504,779638,136331
BC00370=283446,773989,34490
BC00371=283446,773989,34489
BC00372=283446,773989,34490
BC00373=283446,773989,7727
BC00374=283446,773989,13251
BC00375=283446,773989,34490
BC00376=288799,761851,159302
BC00377=294036,749978,281401
BC00378=294036,749978,281401
BC00379=294036,749978,281401
BC00380=294036,749978,281401
BC00381=294036,749978,281401
BC00382=293968,721054,280651
BC00383=293812,675994,279822
BC00384=293812,675994,279822
BC00385=293812,675994,279822
BC00386=294036,749978,281401
BC00387=294036,749978,281401
BC00388=294036,749978,281401
BC00389=294036,749978,281401
BC00390=294036,749978,281401
BC00391=294036,749978,281401
BC00392=293968,721054,280651
BC00393=293968,721054,280651
BC00394=293968,721054,280651
BC00395=293968,721054,280651
BC00396=293968,721054,280651
BC00397=293968,721054,280651
BC00398=293812,675994,279822
BC00399=293812,675994,279822
BC00400=293812,675994,279822
BC00401=293812,675994,279822
BC00402=293812,675994,279822
BC00403=293812,675994,279822
BC00404=290827,666220,220171
BC00405=290827,666220,220171
BC00406=290827,666220,220171
BC00407=290827,666220,220171
BC00408=290827,666220,220171
BC00409=290827,666220,220171
BC00410=290827,666220,220171
BC00411=290827,666220,220171
BC00412=398174,666220,222117
BC00413=398174,666220,222117
BC00414=398174,666220,222117
BC00415=398174,666220,222117
BC00416=398174,666220,222117
BC00417=398174,666220,222117
BC00418=398174,666220,222117
BC00419=398174,666221,222115
BC00420=398174,666221,222116
BC00421=398174,666220,222117
BC00422=398174,666220,222117
BC00423=398174,666220,222117
BC00424=398174,666220,160700
BC00425=398174,666220,116225
BC00426=398174,666220,116225
BC00427=398174,666220,116225
BC00428=398174,666220,116225
BC00429=398174,666220,116225
BC00430=398174,666220,116225
BC00431=398174,666220,116225
BC00432=398174,666220,116225
BC00433=398174,666220,116225
BC00434=398174,666220,116225
BC00435=59154,666220,116225
BC00436=59154,666220,116225
BC00437=59154,666220,116225
BC00438=59154,666220,116225
BC00439=59154,666220,116225
BC00440=59154,666220,116225
BC00441=59154,666220,116225
BC00442=59154,666220,116221
BC00443=59154,666220,116221
BC00444=59154,666220,116221
BC00445=66146,666218,182566
BC00446=118464,666204,678996
EC00000=798156,0
EC00001=798156,0
EC00002=798156,0
EC00003=798156,0
EC00004=798156,0
EC00005=798156,0
EC00006=798156,0
EC00007=798156,0
EC00008=798156,0
EC00009=798156,0
EC00010=798156,0
EC00011=798156,0
EC00012=798156,0
EC00013=798156,0
EC00014=798156,0
EC00015=798156,0
EC00016=798156,0
EC00017=798156,0
EC00018=798156,0
EC00019=798156,0
EC00020=798156,0
EC00021=798156,0
EC00022=798156,0
EC00023=798156,0
EC00024=798156,0
EC00025=798156,0
EC00026=798156,0
EC00027=798156,0
EC00028=798156,0
EC00029=798156,0
EC00030=798156,0
EC00031=798156,0
EC00032=798156,0
EC00033=798156,0
EC00034=798156,0
EC00035=798156,0
EC00036=798156,0
EC00037=798156,0
EC00038=798156,0
EC00039=798156,0
EC00040=798156,0
EC00041=798156,0
EC00042=798156,0
EC00043=798156,0
EC00044=798156,0
EC00045=798156,0
EC00046=798156,0
EC00047=798156,0
EC00048=798156,0
EC00049=798156,0
EC00050=798156,0
EC00051=798156,0
EC00052=798156,0
EC00053=798156,0
EC00054=798156,0
EC00055=798156,0
EC00056=798156,0
EC00057=798156,0
EC00058=798156,0
EC00059=798156,0
EC00060=798156,0
EC00061=798156,0
EC00062=798156,0
EC00063=798156,0
EC00064=798156,0
EC00065=798156,0
EC00066=798156,0
EC00067=798156,0
EC00068=798156,0
EC00069=798156,0
EC00070=798156,0
EC00071=798156,0
EC00072=798156,0
EC00073=798156,0
EC00074=798156,0
EC00075=798156,0
EC00076=798156,0
EC00077=798156,0
EC00078=798156,0
EC00079=798156,0
EC00080=798156,0
EC00081=798156,0
EC00082=798156,0
EC00083=798156,0
EC00084=798156,0
EC00085=798156,0
EC00086=798156,0
EC00087=798156,0
EC00088=798156,0
EC00089=798156,0
EC00090=798156,0
EC00091=798156,0
EC00092=798156,0
EC00093=798156,0
EC00094=798156,0
EC00095=798156,0
EC00096=798156,0
EC00097=798156,0
EC00098=798156,0
EC00099=798156,0
EC00100=798156,0
EC00101=798156,0
EC00102=798156,0
EC00103=798156,0
EC00104=798156,0
EC00105=798156,0
EC00106=798156,0
EC00107=798156,0
EC00108=798156,0
EC00109=798156,0
EC00110=798156,0
EC00111=798156,0
EC00112=798156,0
EC00113=798155,1
EC00114=798155,1
EC00115=798155,1
EC00116=798155,1
EC00117=798155,1
EC00118=798156,0
EC00119=798156,0
EC00120=798156,0
EC00121=798156,0
EC00122=798156,0
EC00123=798155,0
EC00124=798155,0
EC00125=798155,0
EC00126=798155,0
EC00127=798155,0
EC00128=798156,0
EC00129=798156,0
EC00130=798156,0
EC00131=798155,1
EC00132=798155,1
EC00133=798156,0
EC00134=798156,0
EC00135=798156,0
EC00136=798156,0
EC00137=798156,0
EC00138=798156,0
EC00139=798156,0
EC00140=798156,0
EC00141=798156,0
EC00142=798156,0
EC00143=798155,1
EC00144=798155,1
EC00145=798156,0
EC00146=798156,0
EC00147=798156,0
EC00148=798156,0
EC00149=798156,0
EC00150=798156,0
EC00151=798156,0
EC00152=798156,0
EC00153=798156,0
EC00154=798156,0
EC00155=798156,0
EC00156=798156,0
EC00157=798156,0
EC00158=798156,0
EC00159=798156,0
EC00160=798156,0
EC00161=798156,0
EC00162=798156,0
EC00163=798156,0
EC00164=798156,0
EC00165=798156,0
EC00166=798156,0
EC00167=798156,0
EC00168=798156,0
EC00169=798156,0
EC00170=798156,0
EC00171=798156,0
EC00172=798156,0
EC00173=798156,0
EC00174=798156,0
EC00175=798156,0
EC00176=798156,0
EC00177=798156,0
EC00178=798156,0
EC00179=798156,0
EC00180=798156,0
EC00181=798156,0
EC00182=798156,0
EC00183=798155,1
EC00184=798156,0
EC00185=798156,0
EC00186=798156,0
EC00187=798156,0
EC00188=798156,0
EC00189=798156,0
EC00190=798156,0
EC00191=798156,0
EC00192=798156,0
EC00193=798156,0
EC00194=798156,0
EC00195=798156,0
EC00196=798156,0
EC00197=798156,0
EC00198=798156,0
EC00199=798155,0
EC00200=798156,0
EC00201=798156,0
EC00202=798156,0
EC00203=798156,0
EC00204=798156,0
EC00205=798156,0
EC00206=798156,0
EC00207=798156,0
EC00208=798156,0
EC00209=798156,0
EC00210=798156,0
EC00211=798156,0
EC00212=798156,0
EC00213=798156,0
EC00214=798156,0
EC00215=798156,0
EC00216=798156,0
EC00217=798156,0
EC00218=798156,0
EC00219=798156,0
EC00220=798156,0
EC00221=798156,0
EC00222=798156,0
EC00223=798156,0
EC00224=798156,0
EC00225=310394,0
EC00226=310394,556475
EC00227=310394,1112951
EC00228=798156,1112951
EC00229=798156,1112951
EC00230=798156,1112951
EC00231=798156,1112951
EC00232=798156,1112951
EC00233=798156,1112951
EC00234=798156,1112951
EC00235=798156,1112951
EC00236=798156,1112951
EC00237=798156,1112951
EC00238=798156,1112951
EC00239=798156,1112951
EC00240=798156,1112951
EC00241=798156,1112951
EC00242=798156,1112951
EC00243=798156,1112951
EC00244=798156,1112951
EC00245=798156,1112951
EC00246=798156,1112951
EC00247=798156,1112951
EC00248=798156,1112951
EC00249=798156,1112951
EC00250=798156,1112951
EC00251=798156,1112951
EC00252=798156,1112951
EC00253=798156,1112951
EC00254=798156,1112951
EC00255=798156,1112951
EC00256=798156,1112951
EC00257=798156,1112951
EC00258=798156,1112951
EC00259=798156,1112951
EC00260=798156,1112951
EC00261=798156,1112951
EC00262=798156,1112951
EC00263=798156,1112951
EC00264=798156,1112951
EC00265=798156,1112951
EC00266=798156,1112951
EC00267=798156,1112951
EC00268=798156,1112951
EC00269=798156,1112951
EC00270=798156,1112951
EC00271=798156,1112951
EC00272=798156,1112951
EC00273=798156,1112951
EC00274=798156,1112951
EC00275=798156,1112951
EC00276=798156,1112951
EC00277=798156,1112951
EC00278=798156,1112951
EC00279=798156,1112951
EC00280=798156,1112951
EC00281=798156,1112951
EC00282=798156,1112951
EC00283=798156,1112951
EC00284=798156,1112951
EC00285=798156,1112951
EC00286=798156,1112951
EC00287=798156,1112951
EC00288=798156,1112951
EC00289=798156,1112951
EC00290=798156,1112951
EC00291=798156,1112951
EC00292=798156,1112951
EC00293=798156,1112951
EC00294=798156,1112951
EC00295=798156,1112951
EC00296=798156,1112951
EC00297=798156,1112951
EC00298=798156,1112951
EC00299=798156,1112951
EC00300=798156,1112951
EC00301=798156,1112951
EC00302=798156,1112951
EC00303=798156,1112951
EC00304=798156,1112951
EC00305=798156,1112951
EC00306=798156,1112951
EC00307=798156,1112951
EC00308=798156,1112951
EC00309=798156,1112951
EC00310=798156,1112951
EC00311=798156,1112951
EC00312=798156,1112951
EC00313=798156,1112951
EC00314=798156,1112951
EC00315=798156,1112951
EC00316=798156,1112951
EC00317=798156,1112951
EC00318=798156,1112951
EC00319=798156,1112951
EC00320=798156,1112951
EC00321=798156,1112951
EC00322=798156,1112951
EC00323=798156,1112951
EC00324=798156,1112951
EC00325=798156,1112951
EC00326=798156,1112950
EC00327=798156,1112950
EC00328=798156,1112950
EC00329=798156,1112950
EC00330=798156,1112950
EC00331=798156,1112951
EC00332=798156,1112951
EC00333=798156,1112951
EC00334=798156,1112951
EC00335=798156,1112951
EC00336=798156,1112951
EC00337=798156,1112951
EC00338=798156,1112951
EC00339=798155,1112950
EC00340=798155,1112950
EC00341=798155,1112950
EC00342=798155,1112950
EC00343=798155,1112950
EC00344=798156,1112951
EC00345=798156,1112951
EC00346=798156,1112951
EC00347=798156,1112951
EC00348=798156,1112951
EC00349=798156,1112951
EC00350=798156,1112951
EC00351=798156,1112951
EC00352=798156,1112951
EC00353=798156,1112951
EC00354=798156,1112951
EC00355=798156,1112951
EC00356=798156,1112951
EC00357=798156,1112951
EC00358=798156,1112951
EC00359=798156,1112951
EC00360=798156,1112951
EC00361=798156,1112951
EC00362=798156,1112951
EC00363=798156,1112951
EC00364=798156,1112951
EC00365=798156,1112951
EC00366=798156,1112951
EC00367=798155,1112950
EC00368=798156,1112951
EC00369=798155,1112950
EC00370=798155,1112950
EC00371=798156,1112951
EC00372=798156,1112951
EC00373=798156,1112951
EC00374=798156,1112951
EC00375=798156,1112951
EC00376=798156,1112951
EC00377=798156,1112951
EC00378=798156,1112951
EC00379=798156,1112951
EC00380=798156,1112951
EC00381=798156,1112951
EC00382=798156,1112951
EC00383=798156,1112951
EC00384=798156,1112951
EC00385=798156,1112951
EC00386=798156,1112951
EC00387=798156,1112951
EC00388=798156,1112951
EC00389=798156,1112951
EC00390=798156,1112951
EC00391=798156,1112951
EC00392=798156,1112951
EC00393=798156,1112951
EC00394=798156,1112951
EC00395=798156,1112951
EC00396=798156,1112951
EC00397=798156,1112951
EC00398=798156,1112951
EC00399=798156,1112951
EC00400=798156,1112951
EC00401=798156,1112951
EC00402=798156,1112951
EC00403=798156,1112951
EC00404=798156,1112951
EC00405=798156,1112951
EC00406=798156,1112951
EC00407=798156,1112951
EC00408=798156,1112951
EC00409=798156,1112951
EC00410=798156,1112951
EC00411=798156,1112951
EC00412=798156,1112951
EC00413=798156,1112951
EC00414=798156,1112951
EC00415=798155,1112950
EC00416=798155,1112950
EC00417=798156,1112951
EC00418=798156,1112951
EC00419=798156,1112951
EC00420=798156,1112951
EC00421=798156,1112951
EC00422=798156,1112951
EC00423=798156,1112951
EC00424=798156,1112951
EC00425=798156,1112951
EC00426=798156,1112951
EC00427=798156,1112951
EC00428=798156,1112951
EC00429=798156,1112951
EC00430=798156,1112951
EC00431=798156,1112951
EC00432=798156,1112951
EC00433=798156,1112951
EC00434=798156,1112951
EC00435=798156,1112951
EC00436=798156,1112951
EC00437=798156,1112951
EC00438=798155,1112950
EC00439=798155,1112950
EC00440=798155,1112950
EC00441=798154,1112948
EC00442=798156,1112951
///POSTYPE BASE
///RECTAN
///RCONF 0,0,0,0,0,0,0,0,0,0,0,0,0,0,0,0,0,0,0,0,0,0,0,0
P00006=0.222,-3.123,-1.508,0.0000,0.0000,0.0000
P00021=-0.225,-6.128,-0.405,0.0000,0.0000,0.0000
P00022=0.222,-3.123,-1.508,0.0000,0.0000,0.0000
P00023=0.143,-0.036,0.682,0.0000,0.0000,0.0000
P00024=0.145,-0.552,1.326,0.0000,0.0000,0.0000
P00025=-2.003,0.006,0.728,0.0000,0.0000,0.0000
P00026=0.562,-0.002,-0.337,0.0000,0.0000,0.0000
P00027=-0.746,0.015,-9.096,0.0000,0.0000,0.0000
P00028=-2.237,-0.018,-7.702,0.0000,0.0000,0.0000
P00029=-2.156,-0.086,-4.681,0.0000,0.0000,0.0000
P00030=5.926,-4.294,-1.390,0.0000,0.0000,0.0000
P00031=1.853,-0.001,-1.549,0.0000,0.0000,0.0000
P00045=-0.068,-0.810,1.603,0.0000,0.0000,0.0000
//INST
///DATE 2024/12/02 11:34
///ATTR SC,RW
///GROUP1 RB1,BS1
///GROUP2 ST1
NOP
'X2_99(90,0)
MOVJ C00000 BC00000 VJ=100.00  +MOVJ EC00000 VJ=100.00
MOVJ C00001 BC00001 VJ=100.00  +MOVJ EC00001 VJ=100.00
'Path S4826
SFTOF3D
MOVJ C00002 BC00002 VJ=100.00  +MOVJ EC00002 VJ=100.00
MOVL C00003 BC00003 V=800.0  +MOVJ EC00003 VJ=100.00
SMOVL C00004 BC00004 V=166.7  +MOVJ EC00004
SREFP 3 C00005 BC00005  +REFP EC00005
CALL JOB:SEARCH-R1-S13D
SET P031 P006
SFTON3D P031
SMOVL C00006 BC00006 V=166.7  +MOVJ EC00006
SREFP 3 C00007 BC00007  +REFP EC00007
CALL JOB:SEARCH-R1-S13D
SET P031 P006
SFTON3D P031
SMOVL C00008 BC00008 V=250.0  +MOVJ EC00008
SMOVL C00009 BC00009 V=250.0  +MOVJ EC00009
SREFP 3 C00010 BC00010  +REFP EC00010
CALL JOB:SEARCH-R1-S13D
SET P031 P006
SFTON3D P031
SMOVL C00011 BC00011 V=250.0  +MOVJ EC00011
MOVL C00012 BC00012 V=1000.0  +MOVJ EC00012 VJ=100.00
'EndPath S4826
MOVJ C00013 BC00013 VJ=100.00  +MOVJ EC00013 VJ=100.00
'Path S4869
SFTOF3D
MOVJ C00014 BC00014 VJ=100.00  +MOVJ EC00014 VJ=100.00
MOVL C00015 BC00015 V=800.0  +MOVJ EC00015 VJ=100.00
SMOVL C00016 BC00016 V=250.0  +MOVJ EC00016
SREFP 3 C00017 BC00017  +REFP EC00017
CALL JOB:SEARCH-R1-S13D
SET P030 P006
SFTON3D P030
SMOVL C00018 BC00018 V=166.7  +MOVJ EC00018
SMOVL C00019 BC00019 V=250.0  +MOVJ EC00019
SMOVL C00020 BC00020 V=250.0  +MOVJ EC00020
SMOVL C00021 BC00021 V=166.7  +MOVJ EC00021
SREFP 3 C00022 BC00022  +REFP EC00022
CALL JOB:SEARCH-R1-S13D
SET P030 P006
SFTON3D P030
SMOVL C00023 BC00023 V=250.0  +MOVJ EC00023
MOVL C00024 BC00024 V=1000.0  +MOVJ EC00024 VJ=100.00
'EndPath S4869
'Path S4870
SFTOF3D
MOVJ C00025 BC00025 VJ=100.00  +MOVJ EC00025 VJ=100.00
SMOVL C00026 BC00026 V=1000.0  +MOVJ EC00026
SMOVL C00027 BC00027 V=250.0  +MOVJ EC00027
SREFP 3 C00028 BC00028  +REFP EC00028
CALL JOB:SEARCH-R1-S13D
SET P029 P006
SFTON3D P029
SMOVL C00029 BC00029 V=250.0  +MOVJ EC00029
SMOVL C00030 BC00030 V=1000.0  +MOVJ EC00030
SMOVL C00031 BC00031 V=250.0  +MOVJ EC00031
SREFP 3 C00032 BC00032  +REFP EC00032
CALL JOB:SEARCH-R1-S13D
SET P029 P006
SFTON3D P029
SMOVL C00033 BC00033 V=250.0  +MOVJ EC00033
MOVL C00034 BC00034 V=1000.0  +MOVJ EC00034 VJ=100.00
'EndPath S4870
'Path S4823
SFTOF3D
MOVJ C00035 BC00035 VJ=100.00  +MOVJ EC00035 VJ=100.00
SMOVL C00036 BC00036 V=1000.0  +MOVJ EC00036
SMOVL C00037 BC00037 V=166.7  +MOVJ EC00037
SREFP 3 C00038 BC00038  +REFP EC00038
CALL JOB:SEARCH-R1-S13D
SET P028 P006
SFTON3D P028
SMOVL C00039 BC00039 V=250.0  +MOVJ EC00039
SMOVL C00040 BC00040 V=250.0  +MOVJ EC00040
SMOVL C00041 BC00041 V=250.0  +MOVJ EC00041
SREFP 3 C00042 BC00042  +REFP EC00042
CALL JOB:SEARCH-R1-S13D
SET P028 P006
SFTON3D P028
MOVL C00043 BC00043 V=1000.0  +MOVJ EC00043 VJ=100.00
SFTOF3D
SMOVL C00044 BC00044 V=1200.0  +MOVJ EC00044
SMOVL C00045 BC00045 V=1200.0  +MOVJ EC00045
SMOVL C00046 BC00046 V=166.7  +MOVJ EC00046
SREFP 3 C00047 BC00047  +REFP EC00047
CALL JOB:SEARCH-R1-S13D
SET P045 P006
SFTON3D P045
SMOVL C00048 BC00048 V=166.7  +MOVJ EC00048
SMOVL C00049 BC00049 V=800.0  +MOVJ EC00049
SMOVL C00050 BC00050 V=166.7  +MOVJ EC00050
SREFP 3 C00051 BC00051  +REFP EC00051
CALL JOB:SEARCH-R1-S13D
SET P045 P006
SFTON3D P045
SMOVL C00052 BC00052 V=166.7  +MOVJ EC00052
SMOVL C00053 BC00053 V=800.0  +MOVJ EC00053
SMOVL C00054 BC00054 V=800.0  +MOVJ EC00054
SMOVL C00055 BC00055 V=166.7  +MOVJ EC00055
SREFP 3 C00056 BC00056  +REFP EC00056
CALL JOB:SEARCH-R1-S13D
SET P045 P006
SFTON3D P045
SMOVL C00057 BC00057 V=250.0  +MOVJ EC00057
SMOVL C00058 BC00058 V=1200.0  +MOVJ EC00058
SFTOF3D
SMOVL C00059 BC00059 V=1200.0  +MOVJ EC00059
SMOVL C00060 BC00060 V=1200.0  +MOVJ EC00060
'EndPath S4823
'Path S4871
SFTOF3D
COMM MOVJ C00061 BC00061 VJ=100.00  +MOVJ EC00061 VJ=100.00
COMM MOVL C00062 BC00062 V=500.0  +MOVJ EC00062 VJ=100.00
COMM SMOVL C00063 BC00063 V=166.7  +MOVJ EC00063
COMM SREFP 3 C00064 BC00064  +REFP EC00064
COMM CALL JOB:SEARCH-R1-S13D
COMM SET P027 P006
COMM SFTON3D P027
COMM SMOVL C00065 BC00065 V=250.0  +MOVJ EC00065
COMM SMOVL C00066 BC00066 V=166.7  +MOVJ EC00066
COMM SREFP 3 C00067 BC00067  +REFP EC00067
COMM CALL JOB:SEARCH-R1-S13D
COMM SET P027 P006
COMM SFTON3D P027
COMM SMOVL C00068 BC00068 V=250.0  +MOVJ EC00068
COMM MOVL C00069 BC00069 V=1000.0  +MOVJ EC00069 VJ=100.00
COMM 'EndPath S4871
COMM 'Path S4872
COMM SFTOF3D
COMM MOVJ C00070 BC00070 VJ=100.00  +MOVJ EC00070 VJ=100.00
COMM MOVL C00071 BC00071 V=500.0  +MOVJ EC00071 VJ=100.00
COMM SMOVL C00072 BC00072 V=166.7  +MOVJ EC00072
COMM SREFP 3 C00073 BC00073  +REFP EC00073
COMM CALL JOB:SEARCH-R1-S13D
COMM SET P026 P006
COMM SFTON3D P026
COMM SMOVL C00074 BC00074 V=250.0  +MOVJ EC00074
COMM SMOVL C00075 BC00075 V=166.7  +MOVJ EC00075
COMM SREFP 3 C00076 BC00076  +REFP EC00076
COMM CALL JOB:SEARCH-R1-S13D
COMM SET P026 P006
COMM SFTON3D P026
COMM SMOVL C00077 BC00077 V=800.0  +MOVJ EC00077
COMM MOVL C00078 BC00078 V=1000.0  +MOVJ EC00078 VJ=100.00
COMM 'EndPath S4872
COMM 'Path S4820
COMM SFTOF3D
COMM MOVJ C00079 BC00079 VJ=100.00  +MOVJ EC00079 VJ=100.00
COMM MOVL C00080 BC00080 V=500.0  +MOVJ EC00080 VJ=100.00
COMM SMOVL C00081 BC00081 V=166.7  +MOVJ EC00081
COMM SREFP 3 C00082 BC00082  +REFP EC00082
COMM CALL JOB:SEARCH-R1-S13D
COMM SET P025 P006
COMM SFTON3D P025
COMM SMOVL C00083 BC00083 V=250.0  +MOVJ EC00083
COMM SMOVL C00084 BC00084 V=166.7  +MOVJ EC00084
COMM SREFP 3 C00085 BC00085  +REFP EC00085
COMM CALL JOB:SEARCH-R1-S13D
COMM SET P025 P006
COMM SFTON3D P025
COMM SMOVL C00086 BC00086 V=250.0  +MOVJ EC00086
COMM MOVL C00087 BC00087 V=1000.0  +MOVJ EC00087 VJ=100.00
COMM 'EndPath S4820
MOVJ C00088 BC00088 VJ=100.00  +MOVJ EC00088 VJ=100.00
MOVJ C00089 BC00089 VJ=100.00  +MOVJ EC00089 VJ=100.00
'Path S4819 (for W4811)
SFTOF3D
MOVJ C00090 BC00090 VJ=100.00  +MOVJ EC00090 VJ=100.00
MOVL C00091 BC00091 V=666.7  +MOVJ EC00091 VJ=100.00
SMOVL C00092 BC00092 V=166.7  +MOVJ EC00092
SREFP 3 C00093 BC00093  +REFP EC00093
CALL JOB:SEARCH-R1-S13D
SET P024 P006
SFTON3D P024
SMOVL C00094 BC00094 V=166.7  +MOVJ EC00094
SREFP 3 C00095 BC00095  +REFP EC00095
CALL JOB:SEARCH-R1-S13D
SET P024 P006
SFTON3D P024
SMOVL C00096 BC00096 V=166.7  +MOVJ EC00096
MOVL C00097 BC00097 V=1000.0  +MOVJ EC00097 VJ=100.00
'EndPath S4819 (for W4811)
'Path S4818 (for W4811)
SFTOF3D
MOVJ C00098 BC00098 VJ=100.00  +MOVJ EC00098 VJ=100.00
MOVL C00099 BC00099 V=500.0  +MOVJ EC00099 VJ=100.00
SMOVL C00100 BC00100 V=166.7  +MOVJ EC00100
SREFP 3 C00101 BC00101  +REFP EC00101
CALL JOB:SEARCH-R1-S13D
SET P023 P006
SFTON3D P023
SMOVL C00102 BC00102 V=166.7  +MOVJ EC00102
SMOVL C00103 BC00103 V=166.7  +MOVJ EC00103
SREFP 3 C00104 BC00104  +REFP EC00104
CALL JOB:SEARCH-R1-S13D
SET P023 P006
SFTON3D P023
SMOVL C00105 BC00105 V=166.7  +MOVJ EC00105
MOVL C00106 BC00106 V=1000.0  +MOVJ EC00106 VJ=100.00
'EndPath S4818 (for W4811)
MOVJ C00107 BC00107 VJ=100.00  +MOVJ EC00107 VJ=100.00
MOVJ C00108 BC00108 VJ=100.00  +MOVJ EC00108 VJ=100.00
MOVJ C00109 BC00109 VJ=100.00  +MOVJ EC00109 VJ=100.00
'Path S4816 (for W4808)
SFTOF3D
MOVJ C00110 BC00110 VJ=100.00  +MOVJ EC00110 VJ=100.00
MOVL C00111 BC00111 V=500.0  +MOVJ EC00111 VJ=100.00
SMOVL C00112 BC00112 V=166.7  +MOVJ EC00112
SREFP 3 C00113 BC00113  +REFP EC00113
CALL JOB:SEARCH-R1-S13D
SET P021 P006
SFTON3D P021
SMOVL C00114 BC00114 V=166.7  +MOVJ EC00114
SMOVL C00115 BC00115 V=166.7  +MOVJ EC00115
SREFP 3 C00116 BC00116  +REFP EC00116
CALL JOB:SEARCH-R1-S13D
SET P021 P006
SFTON3D P021
SMOVL C00117 BC00117 V=166.7  +MOVJ EC00117
MOVL C00118 BC00118 V=1000.0  +MOVJ EC00118 VJ=100.00
'EndPath S4816 (for W4808)
MOVJ C00119 BC00119 VJ=100.00  +MOVJ EC00119 VJ=100.00
'Path S4817 (for W4808)
SFTOF3D
MOVJ C00120 BC00120 VJ=100.00  +MOVJ EC00120 VJ=100.00
MOVL C00121 BC00121 V=500.0  +MOVJ EC00121 VJ=100.00
SMOVL C00122 BC00122 V=166.7  +MOVJ EC00122
SREFP 3 C00123 BC00123  +REFP EC00123
CALL JOB:SEARCH-R1-S13D
SET P022 P006
SFTON3D P022
SMOVL C00124 BC00124 V=166.7  +MOVJ EC00124
SMOVL C00125 BC00125 V=166.7  +MOVJ EC00125
SREFP 3 C00126 BC00126  +REFP EC00126
CALL JOB:SEARCH-R1-S13D
SET P022 P006
SFTON3D P022
SMOVL C00127 BC00127 V=166.7  +MOVJ EC00127
'EndPath S4817 (for W4808)
'Path W4808
SFTOF3D
SFTON3D P022
MOVJ C00128 BC00128 VJ=100.00  +MOVJ EC00128 VJ=100.00
SMOVL C00129 BC00129 V=800.0  +MOVJ EC00129
REFP 1 RB1 C00130 BC00130
REFP 1 RB1 C00131 BC00131
SMOVL C00132 BC00132 V=150.0 PL=0  +MOVJ EC00130
SWVON WEV#(100)
MACRO1 MJ#(0) ARGF21
ARCON
SMOVL C00133 BC00133 V=8.3  +MOVJ EC00131
SMOVL C00134 BC00134 V=8.3  +MOVJ EC00132
SFTON3D P021
SMOVL C00135 BC00135 V=8.3  +MOVJ EC00133
SMOVL C00136 BC00136 V=8.3  +MOVJ EC00134
ARCOF
SWVOF
SMOVL C00137 BC00137 V=800.0  +MOVJ EC00135
SMOVL C00138 BC00138 V=1000.0  +MOVJ EC00136
SFTOF3D
'EndPath W4808
MOVJ C00139 BC00139 VJ=100.00  +MOVJ EC00137 VJ=100.00
MOVJ C00140 BC00140 VJ=100.00  +MOVJ EC00138 VJ=100.00
MOVJ C00141 BC00141 VJ=100.00  +MOVJ EC00139 VJ=100.00
MOVJ C00142 BC00142 VJ=100.00  +MOVJ EC00140 VJ=100.00
MOVJ C00143 BC00143 VJ=100.00  +MOVJ EC00141 VJ=100.00
'Path W4811
SFTOF3D
SFTON3D P024
MOVJ C00144 BC00144 VJ=100.00  +MOVJ EC00142 VJ=100.00
SMOVL C00145 BC00145 V=800.0  +MOVJ EC00143
REFP 1 RB1 C00146 BC00146
REFP 2 RB1 C00147 BC00147
SMOVL C00148 BC00148 V=150.0 PL=0  +MOVJ EC00144
MACRO1 MJ#(0) ARGF9
SWVON WEV#(100)
ARCON
SFTON3D P023
SMOVL C00149 BC00149 V=8.3  +MOVJ EC00145
ARCOF
SWVOF
SMOVL C00150 BC00150 V=800.0  +MOVJ EC00146
SMOVL C00151 BC00151 V=1000.0  +MOVJ EC00147
SFTOF3D
'EndPath W4811
'
MOVJ C00152 BC00152 VJ=100.00  +MOVJ EC00148 VJ=100.00
MOVJ C00153 BC00153 VJ=100.00  +MOVJ EC00149 VJ=100.00
MOVJ C00154 BC00154 VJ=100.00  +MOVJ EC00150 VJ=100.00
'Path W4873
SFTOF3D
COMM SFTON3D P025
COMM MOVJ C00155 BC00155 VJ=100.00  +MOVJ EC00151 VJ=100.00
COMM SMOVL C00156 BC00156 V=800.0  +MOVJ EC00152
COMM SMOVL C00157 BC00157 V=150.0 PL=0  +MOVJ EC00153
COMM MACRO1 MJ#(0) ARGF14
COMM ARCON
COMM SMOVL C00158 BC00158 V=10.0  +MOVJ EC00154
COMM SMOVL C00159 BC00159 V=10.8  +MOVJ EC00155
COMM SFTON3D P026
COMM SMOVL C00160 BC00160 V=10.8  +MOVJ EC00156
COMM SFTON3D P027
COMM SMOVL C00161 BC00161 V=10.8  +MOVJ EC00157
COMM ARCOF
COMM SMOVL C00162 BC00162 V=800.0  +MOVJ EC00158
COMM SMOVL C00163 BC00163 V=1000.0  +MOVJ EC00159
COMM SFTOF3D
COMM SFTON3D P025
COMM MOVJ C00164 BC00164 VJ=100.00  +MOVJ EC00160 VJ=100.00
COMM SMOVL C00165 BC00165 V=800.0  +MOVJ EC00161
COMM SMOVL C00166 BC00166 V=150.0 PL=0  +MOVJ EC00162
COMM MACRO1 MJ#(0) ARGF14
COMM ARCON
COMM SMOVL C00167 BC00167 V=10.8  +MOVJ EC00163
COMM ARCON
COMM SMOVL C00168 BC00168 V=10.0  +MOVJ EC00164
COMM ARCOF
COMM SMOVL C00169 BC00169 V=800.0  +MOVJ EC00165
COMM SMOVL C00170 BC00170 V=1000.0  +MOVJ EC00166
COMM SFTOF3D
COMM 'EndPath W4873
COMM 'Path W4874
COMM SFTOF3D
COMM SFTON3D P026
COMM MOVJ C00171 BC00171 VJ=100.00  +MOVJ EC00167 VJ=100.00
COMM SMOVL C00172 BC00172 V=800.0  +MOVJ EC00168
COMM SMOVL C00173 BC00173 V=150.0 PL=0  +MOVJ EC00169
COMM ARCON
COMM SMOVL C00174 BC00174 V=10.8  +MOVJ EC00170
COMM ARCOF
COMM SMOVL C00175 BC00175 V=800.0  +MOVJ EC00171
COMM SMOVL C00176 BC00176 V=1000.0  +MOVJ EC00172
COMM SFTOF3D
COMM 'EndPath W4874
COMM 'Path W4875
COMM SFTOF3D
COMM SFTON3D P027
COMM MOVJ C00177 BC00177 VJ=100.00  +MOVJ EC00173 VJ=100.00
COMM SMOVL C00178 BC00178 V=800.0  +MOVJ EC00174
COMM SMOVL C00179 BC00179 V=150.0 PL=0  +MOVJ EC00175
COMM ARCON
COMM SMOVL C00180 BC00180 V=10.8  +MOVJ EC00176
COMM ARCOF
COMM SMOVL C00181 BC00181 V=800.0  +MOVJ EC00177
COMM SMOVL C00182 BC00182 V=1000.0  +MOVJ EC00178
COMM SFTOF3D
'EndPath W4875
'Path W4876
SFTOF3D
SFTON3D P028
MOVJ C00183 BC00183 VJ=100.00  +MOVJ EC00179 VJ=100.00
SMOVL C00184 BC00184 V=800.0  +MOVJ EC00180
SMOVL C00185 BC00185 V=150.0 PL=0  +MOVJ EC00181
ARCON
SFTON3D P029
SMOVL C00186 BC00186 V=11.7  +MOVJ EC00182
SMOVL C00187 BC00187 V=11.7  +MOVJ EC00183
ARCOF
SMOVL C00188 BC00188 V=800.0  +MOVJ EC00184
SMOVL C00189 BC00189 V=1000.0  +MOVJ EC00185
SFTOF3D
'EndPath W4876
MOVJ C00190 BC00190 VJ=100.00  +MOVJ EC00186 VJ=100.00
MOVJ C00191 BC00191 VJ=100.00  +MOVJ EC00187 VJ=100.00
MOVJ C00192 BC00192 VJ=100.00  +MOVJ EC00188 VJ=100.00
'Path W4877
SFTOF3D
SFTON3D P030
MOVJ C00193 BC00193 VJ=100.00  +MOVJ EC00189 VJ=100.00
SMOVL C00194 BC00194 V=800.0  +MOVJ EC00190
SMOVL C00195 BC00195 V=150.0 PL=0  +MOVJ EC00191
ARCON
SMOVL C00196 BC00196 V=10.8  +MOVJ EC00192
SMOVL C00197 BC00197 V=10.8  +MOVJ EC00193
SMOVL C00198 BC00198 V=10.0  +MOVJ EC00194
ARCOF
SMOVL C00199 BC00199 V=800.0  +MOVJ EC00195
SMOVL C00200 BC00200 V=1000.0  +MOVJ EC00196
SFTOF3D
'EndPath W4877
MOVJ C00201 BC00201 VJ=100.00  +MOVJ EC00197 VJ=100.00
MOVJ C00202 BC00202 VJ=100.00  +MOVJ EC00198 VJ=100.00
'Path W4878
SFTOF3D
SFTON3D P031
MOVJ C00203 BC00203 VJ=100.00  +MOVJ EC00199 VJ=100.00
SMOVL C00204 BC00204 V=800.0  +MOVJ EC00200
MACRO1 MJ#(0) ARGF9
SMOVL C00205 BC00205 V=150.0 PL=0  +MOVJ EC00201
ARCON
SMOVL C00206 BC00206 V=10.0 PL=0  +MOVJ EC00202
ARCON
SWVON WEV#(101)
SMOVL C00207 BC00207 V=8.3  +MOVJ EC00203
SMOVL C00208 BC00208 V=8.3  +MOVJ EC00204
SWVOF
SFTON3D P030
MACRO1 MJ#(0) ARGF14
SMOVL C00209 BC00209 V=10.0  +MOVJ EC00205
ARCOF
SMOVL C00210 BC00210 V=800.0  +MOVJ EC00206
SMOVL C00211 BC00211 V=1000.0  +MOVJ EC00207
SFTOF3D
'EndPath W4878
MOVJ C00212 BC00212 VJ=100.00  +MOVJ EC00208 VJ=100.00
MOVJ C00213 BC00213 VJ=100.00  +MOVJ EC00209 VJ=100.00
MOVJ C00214 BC00214 VJ=100.00  +MOVJ EC00210 VJ=100.00
SFTON3D P045
MACRO1 MJ#(0) ARGF6
SMOVL C00215 BC00215 V=166.7  +MOVJ EC00211
ARCON
SMOVL C00216 BC00216 V=10.0  +MOVJ EC00212
ARCOF
SMOVL C00217 BC00217 V=166.7  +MOVJ EC00213
SMOVL C00218 BC00218 V=166.7  +MOVJ EC00214
SMOVL C00219 BC00219 V=166.7  +MOVJ EC00215
ARCON
SMOVL C00220 BC00220 V=11.7  +MOVJ EC00216
ARCOF
SMOVL C00221 BC00221 V=250.0  +MOVJ EC00217
MOVJ C00222 BC00222 VJ=100.00  +MOVJ EC00218 VJ=100.00
MOVJ C00223 BC00223 VJ=100.00  +MOVJ EC00219 VJ=100.00
MOVJ C00224 BC00224 VJ=100.00  +MOVJ EC00220 VJ=100.00
SMOVL C00225 BC00225 V=166.7  +MOVJ EC00221
ARCON
SMOVL C00226 BC00226 V=11.7  +MOVJ EC00222
ARCOF
SMOVL C00227 BC00227 V=800.0  +MOVJ EC00223
SFTOF3D
MOVJ C00228 BC00228 VJ=100.00  +MOVJ EC00224 VJ=100.00
MOVJ C00229 BC00229 VJ=100.00  +MOVJ EC00225 VJ=100.00
MOVJ C00230 BC00230 VJ=100.00  +MOVJ EC00226 VJ=100.00
MOVJ C00231 BC00231 VJ=100.00  +MOVJ EC00227 VJ=100.00
MOVJ C00232 BC00232 VJ=100.00  +MOVJ EC00228 VJ=100.00
CALL JOB:CLEAN-R1_KM_NEW
'
'
'
'
'
'
'Path S4829
SFTOF3D
MOVJ C00233 BC00233 VJ=100.00  +MOVJ EC00229 VJ=100.00
MOVL C00234 BC00234 V=666.7  +MOVJ EC00230 VJ=100.00
SMOVL C00235 BC00235 V=166.7  +MOVJ EC00231
SREFP 3 C00236 BC00236  +REFP EC00232
CALL JOB:SEARCH-R1-S13D
SET P031 P006
SFTON3D P031
SMOVL C00237 BC00237 V=166.7  +MOVJ EC00233
SREFP 3 C00238 BC00238  +REFP EC00234
CALL JOB:SEARCH-R1-S13D
SET P031 P006
SFTON3D P031
SMOVL C00239 BC00239 V=166.7  +MOVJ EC00235
SMOVL C00240 BC00240 V=666.7  +MOVJ EC00236
SMOVL C00241 BC00241 V=166.7  +MOVJ EC00237
SREFP 3 C00242 BC00242  +REFP EC00238
CALL JOB:SEARCH-R1-S13D
SET P031 P006
SFTON3D P031
SMOVL C00243 BC00243 V=166.7  +MOVJ EC00239
'EndPath S4829
MOVJ C00244 BC00244 VJ=100.00  +MOVJ EC00240 VJ=100.00
'Path S4830
SFTOF3D
MOVJ C00245 BC00245 VJ=100.00  +MOVJ EC00241 VJ=100.00
SMOVL C00246 BC00246 V=666.7  +MOVJ EC00242
SMOVL C00247 BC00247 V=166.7  +MOVJ EC00243
SREFP 3 C00248 BC00248  +REFP EC00244
CALL JOB:SEARCH-R1-S13D
SET P030 P006
SFTON3D P030
SMOVL C00249 BC00249 V=166.7  +MOVJ EC00245
SMOVL C00250 BC00250 V=666.7  +MOVJ EC00246
SMOVL C00251 BC00251 V=166.7  +MOVJ EC00247
SREFP 3 C00252 BC00252  +REFP EC00248
CALL JOB:SEARCH-R1-S13D
SET P030 P006
SFTON3D P030
SMOVL C00253 BC00253 V=250.0  +MOVJ EC00249
MOVL C00254 BC00254 V=1000.0  +MOVJ EC00250 VJ=100.00
'EndPath S4830
'Path S4831
SFTOF3D
MOVJ C00255 BC00255 VJ=100.00  +MOVJ EC00251 VJ=100.00
SMOVL C00256 BC00256 V=666.7  +MOVJ EC00252
SMOVL C00257 BC00257 V=166.7  +MOVJ EC00253
SREFP 3 C00258 BC00258  +REFP EC00254
CALL JOB:SEARCH-R1-S13D
SET P029 P006
SFTON3D P029
SMOVL C00259 BC00259 V=166.7  +MOVJ EC00255
SMOVL C00260 BC00260 V=666.7  +MOVJ EC00256
SMOVL C00261 BC00261 V=166.7  +MOVJ EC00257
SREFP 3 C00262 BC00262  +REFP EC00258
CALL JOB:SEARCH-R1-S13D
SET P029 P006
SFTON3D P029
SMOVL C00263 BC00263 V=250.0  +MOVJ EC00259
MOVL C00264 BC00264 V=1000.0  +MOVJ EC00260 VJ=100.00
'EndPath S4831
'Path S4832
SFTOF3D
SMOVL C00265 BC00265 V=1200.0  +MOVJ EC00261
SMOVL C00266 BC00266 V=1000.0  +MOVJ EC00262
SMOVL C00267 BC00267 V=166.7  +MOVJ EC00263
SREFP 3 C00268 BC00268  +REFP EC00264
CALL JOB:SEARCH-R1-S13D
SET P045 P006
SFTON3D P045
SMOVL C00269 BC00269 V=166.7  +MOVJ EC00265
SMOVL C00270 BC00270 V=333.3  +MOVJ EC00266
SMOVL C00271 BC00271 V=166.7  +MOVJ EC00267
SREFP 3 C00272 BC00272  +REFP EC00268
CALL JOB:SEARCH-R1-S13D
SET P045 P006
SFTON3D P045
SMOVL C00273 BC00273 V=166.7  +MOVJ EC00269
SMOVL C00274 BC00274 V=800.0  +MOVJ EC00270
SMOVL C00275 BC00275 V=166.7  +MOVJ EC00271
SREFP 3 C00276 BC00276  +REFP EC00272
CALL JOB:SEARCH-R1-S13D
SET P045 P006
SFTON3D P045
SMOVL C00277 BC00277 V=166.7  +MOVJ EC00273
SFTOF3D
SMOVL C00278 BC00278 V=1000.0  +MOVJ EC00274
SMOVL C00279 BC00279 V=1200.0  +MOVJ EC00275
SMOVL C00280 BC00280 V=666.7  +MOVJ EC00276
SMOVL C00281 BC00281 V=166.7  +MOVJ EC00277
SREFP 3 C00282 BC00282  +REFP EC00278
CALL JOB:SEARCH-R1-S13D
SET P028 P006
SFTON3D P028
SMOVL C00283 BC00283 V=166.7  +MOVJ EC00279
SMOVL C00284 BC00284 V=666.7  +MOVJ EC00280
SMOVL C00285 BC00285 V=166.7  +MOVJ EC00281
SREFP 3 C00286 BC00286  +REFP EC00282
CALL JOB:SEARCH-R1-S13D
SET P028 P006
SFTON3D P028
SMOVL C00287 BC00287 V=166.7  +MOVJ EC00283
MOVL C00288 BC00288 V=1000.0  +MOVJ EC00284 VJ=100.00
'EndPath S4832
MOVJ C00289 BC00289 VJ=100.00  +MOVJ EC00285 VJ=100.00
'Path S4833
SFTOF3D
COMM MOVJ C00290 BC00290 VJ=100.00  +MOVJ EC00286 VJ=100.00
COMM MOVL C00291 BC00291 V=666.7  +MOVJ EC00287 VJ=100.00
COMM SMOVL C00292 BC00292 V=166.7  +MOVJ EC00288
COMM SREFP 3 C00293 BC00293  +REFP EC00289
COMM CALL JOB:SEARCH-R1-S13D
COMM SET P027 P006
COMM SFTON3D P027
COMM SMOVL C00294 BC00294 V=166.7  +MOVJ EC00290
COMM SMOVL C00295 BC00295 V=166.7  +MOVJ EC00291
COMM SREFP 3 C00296 BC00296  +REFP EC00292
COMM CALL JOB:SEARCH-R1-S13D
COMM SET P027 P006
COMM SFTON3D P027
COMM SMOVL C00297 BC00297 V=166.7  +MOVJ EC00293
COMM MOVL C00298 BC00298 V=1000.0  +MOVJ EC00294 VJ=100.00
COMM 'EndPath S4833
COMM 'Path S4834
COMM SFTOF3D
COMM MOVJ C00299 BC00299 VJ=100.00  +MOVJ EC00295 VJ=100.00
COMM MOVL C00300 BC00300 V=666.7  +MOVJ EC00296 VJ=100.00
COMM SMOVL C00301 BC00301 V=166.7  +MOVJ EC00297
COMM SREFP 3 C00302 BC00302  +REFP EC00298
COMM CALL JOB:SEARCH-R1-S13D
COMM SET P026 P006
COMM SFTON3D P026
COMM SMOVL C00303 BC00303 V=166.7  +MOVJ EC00299
COMM SMOVL C00304 BC00304 V=166.7  +MOVJ EC00300
COMM SREFP 3 C00305 BC00305  +REFP EC00301
COMM CALL JOB:SEARCH-R1-S13D
COMM SET P026 P006
COMM SFTON3D P026
COMM SMOVL C00306 BC00306 V=166.7  +MOVJ EC00302
COMM 'EndPath S4834
COMM 'Path S4835
COMM SFTOF3D
COMM MOVJ C00307 BC00307 VJ=100.00  +MOVJ EC00303 VJ=100.00
COMM MOVL C00308 BC00308 V=666.7  +MOVJ EC00304 VJ=100.00
COMM SMOVL C00309 BC00309 V=166.7  +MOVJ EC00305
COMM SREFP 3 C00310 BC00310  +REFP EC00306
COMM CALL JOB:SEARCH-R1-S13D
COMM SET P025 P006
COMM SFTON3D P025
COMM SMOVL C00311 BC00311 V=166.7  +MOVJ EC00307
COMM SMOVL C00312 BC00312 V=166.7  +MOVJ EC00308
COMM SREFP 3 C00313 BC00313  +REFP EC00309
COMM CALL JOB:SEARCH-R1-S13D
COMM SET P025 P006
COMM SFTON3D P025
COMM SMOVL C00314 BC00314 V=166.7  +MOVJ EC00310
COMM MOVL C00315 BC00315 V=1000.0  +MOVJ EC00311 VJ=100.00
COMM 'EndPath S4835
MOVJ C00316 BC00316 VJ=100.00  +MOVJ EC00312 VJ=100.00
MOVJ C00317 BC00317 VJ=100.00  +MOVJ EC00313 VJ=100.00
'Path S4836 (for W4841)
SFTOF3D
MOVJ C00318 BC00318 VJ=100.00  +MOVJ EC00314 VJ=100.00
MOVL C00319 BC00319 V=666.7  +MOVJ EC00315 VJ=100.00
SMOVL C00320 BC00320 V=166.7  +MOVJ EC00316
SREFP 3 C00321 BC00321  +REFP EC00317
CALL JOB:SEARCH-R1-S13D
SET P024 P006
SFTON3D P024
SMOVL C00322 BC00322 V=166.7  +MOVJ EC00318
SMOVL C00323 BC00323 V=166.7  +MOVJ EC00319
SREFP 3 C00324 BC00324  +REFP EC00320
CALL JOB:SEARCH-R1-S13D
SET P024 P006
SFTON3D P024
SMOVL C00325 BC00325 V=166.7  +MOVJ EC00321
MOVL C00326 BC00326 V=1000.0  +MOVJ EC00322 VJ=100.00
'EndPath S4836 (for W4841)
'Path S4837 (for W4841)
SFTOF3D
MOVJ C00327 BC00327 VJ=100.00  +MOVJ EC00323 VJ=100.00
MOVL C00328 BC00328 V=666.7  +MOVJ EC00324 VJ=100.00
SMOVL C00329 BC00329 V=166.7  +MOVJ EC00325
SREFP 3 C00330 BC00330  +REFP EC00326
CALL JOB:SEARCH-R1-S13D
SET P023 P006
SFTON3D P023
SMOVL C00331 BC00331 V=166.7  +MOVJ EC00327
SMOVL C00332 BC00332 V=166.7  +MOVJ EC00328
SREFP 3 C00333 BC00333  +REFP EC00329
CALL JOB:SEARCH-R1-S13D
SET P023 P006
SFTON3D P023
SMOVL C00334 BC00334 V=166.7  +MOVJ EC00330
MOVL C00335 BC00335 V=1000.0  +MOVJ EC00331 VJ=100.00
'EndPath S4837 (for W4841)
MOVJ C00336 BC00336 VJ=100.00  +MOVJ EC00332 VJ=100.00
MOVJ C00337 BC00337 VJ=100.00  +MOVJ EC00333 VJ=100.00
MOVJ C00338 BC00338 VJ=100.00  +MOVJ EC00334 VJ=100.00
MOVJ C00339 BC00339 VJ=100.00  +MOVJ EC00335 VJ=100.00
'Path S4838 (for W4840)
SFTOF3D
MOVJ C00340 BC00340 VJ=100.00  +MOVJ EC00336 VJ=100.00
MOVL C00341 BC00341 V=666.7  +MOVJ EC00337 VJ=100.00
SMOVL C00342 BC00342 V=166.7  +MOVJ EC00338
SREFP 3 C00343 BC00343  +REFP EC00339
CALL JOB:SEARCH-R1-S13D
SET P021 P006
SFTON3D P021
SMOVL C00344 BC00344 V=166.7  +MOVJ EC00340
SMOVL C00345 BC00345 V=166.7  +MOVJ EC00341
SREFP 3 C00346 BC00346  +REFP EC00342
CALL JOB:SEARCH-R1-S13D
SET P021 P006
SFTON3D P021
SMOVL C00347 BC00347 V=166.7  +MOVJ EC00343
MOVL C00348 BC00348 V=1000.0  +MOVJ EC00344 VJ=100.00
'EndPath S4838 (for W4840)
MOVJ C00349 BC00349 VJ=100.00  +MOVJ EC00345 VJ=100.00
'Path S4839 (for W4840)
SFTOF3D
MOVJ C00350 BC00350 VJ=100.00  +MOVJ EC00346 VJ=100.00
MOVL C00351 BC00351 V=666.7  +MOVJ EC00347 VJ=100.00
SMOVL C00352 BC00352 V=166.7  +MOVJ EC00348
SREFP 3 C00353 BC00353  +REFP EC00349
CALL JOB:SEARCH-R1-S13D
SET P022 P006
SFTON3D P022
SMOVL C00354 BC00354 V=166.7  +MOVJ EC00350
SMOVL C00355 BC00355 V=166.7  +MOVJ EC00351
SREFP 3 C00356 BC00356  +REFP EC00352
CALL JOB:SEARCH-R1-S13D
SET P022 P006
SFTON3D P022
SMOVL C00357 BC00357 V=166.7  +MOVJ EC00353
'EndPath S4839 (for W4840)
'Path W4840
SFTOF3D
SFTON3D P022
SMOVL C00358 BC00358 V=800.0  +MOVJ EC00354
SREFP 1 C00359 BC00359  +REFP EC00355
SREFP 2 C00360 BC00360  +REFP EC00356
SMOVL C00361 BC00361 V=150.0 PL=0  +MOVJ EC00357
MACRO1 MJ#(0) ARGF21
ARCON
SWVON WEV#(100)
SMOVL C00362 BC00362 V=8.3  +MOVJ EC00358
SFTON3D P021
SMOVL C00363 BC00363 V=8.3  +MOVJ EC00359
ARCOF
SWVOF
SMOVL C00364 BC00364 V=800.0  +MOVJ EC00360
SMOVL C00365 BC00365 V=1000.0  +MOVJ EC00361
SFTOF3D
'EndPath W4840
MOVJ C00366 BC00366 VJ=100.00  +MOVJ EC00362 VJ=100.00
MOVJ C00367 BC00367 VJ=100.00  +MOVJ EC00363 VJ=100.00
MOVJ C00368 BC00368 VJ=100.00  +MOVJ EC00364 VJ=100.00
MOVJ C00369 BC00369 VJ=100.00  +MOVJ EC00365 VJ=100.00
'Path W4841
SFTOF3D
SFTON3D P024
MOVJ C00370 BC00370 VJ=100.00  +MOVJ EC00366 VJ=100.00
SMOVL C00371 BC00371 V=800.0  +MOVJ EC00367
SMOVL C00372 BC00372 V=150.0 PL=0  +MOVJ EC00368
ARCON
SWVON WEV#(100)
SFTON3D P023
SMOVL C00373 BC00373 V=8.3  +MOVJ EC00369
ARCOF
SWVOF
SMOVL C00374 BC00374 V=800.0  +MOVJ EC00370
SMOVL C00375 BC00375 V=1000.0  +MOVJ EC00371
SFTOF3D
'EndPath W4841
'
MOVJ C00376 BC00376 VJ=100.00  +MOVJ EC00372 VJ=100.00
'Path W4842
SFTOF3D
COMM SFTON3D P025
COMM MOVJ C00377 BC00377 VJ=100.00  +MOVJ EC00373 VJ=100.00
COMM SMOVL C00378 BC00378 V=800.0  +MOVJ EC00374
COMM SMOVL C00379 BC00379 V=150.0 PL=0  +MOVJ EC00375
COMM MACRO1 MJ#(0) ARGF14
COMM ARCON
COMM SMOVL C00380 BC00380 V=10.8  +MOVJ EC00376
COMM SMOVL C00381 BC00381 V=10.8  +MOVJ EC00377
COMM SFTON3D P026
COMM SMOVL C00382 BC00382 V=10.8  +MOVJ EC00378
COMM SFTON3D P027
COMM SMOVL C00383 BC00383 V=10.8  +MOVJ EC00379
COMM ARCOF
COMM SMOVL C00384 BC00384 V=800.0  +MOVJ EC00380
COMM SMOVL C00385 BC00385 V=1000.0  +MOVJ EC00381
COMM SFTOF3D
COMM SFTON3D P025
COMM MOVJ C00386 BC00386 VJ=100.00  +MOVJ EC00382 VJ=100.00
COMM SMOVL C00387 BC00387 V=800.0  +MOVJ EC00383
COMM SMOVL C00388 BC00388 V=150.0 PL=0  +MOVJ EC00384
COMM MACRO1 MJ#(0) ARGF9
COMM ARCON
COMM SMOVL C00389 BC00389 V=12.5  +MOVJ EC00385
COMM ARCOF
COMM SMOVL C00390 BC00390 V=800.0  +MOVJ EC00386
COMM SMOVL C00391 BC00391 V=1000.0  +MOVJ EC00387
COMM SFTOF3D
COMM 'EndPath W4842
COMM 'Path W4843
COMM SFTOF3D
COMM SFTON3D P026
COMM MOVJ C00392 BC00392 VJ=100.00  +MOVJ EC00388 VJ=100.00
COMM SMOVL C00393 BC00393 V=800.0  +MOVJ EC00389
COMM SMOVL C00394 BC00394 V=150.0 PL=0  +MOVJ EC00390
COMM ARCON
COMM SMOVL C00395 BC00395 V=12.5  +MOVJ EC00391
COMM ARCOF
COMM SMOVL C00396 BC00396 V=800.0  +MOVJ EC00392
COMM SMOVL C00397 BC00397 V=1000.0  +MOVJ EC00393
COMM SFTOF3D
COMM 'EndPath W4843
COMM 'Path W4844
COMM SFTOF3D
COMM SFTON3D P027
COMM MOVJ C00398 BC00398 VJ=100.00  +MOVJ EC00394 VJ=100.00
COMM SMOVL C00399 BC00399 V=800.0  +MOVJ EC00395
COMM SMOVL C00400 BC00400 V=150.0 PL=0  +MOVJ EC00396
COMM ARCON
COMM SMOVL C00401 BC00401 V=12.5  +MOVJ EC00397
COMM ARCOF
COMM SMOVL C00402 BC00402 V=800.0  +MOVJ EC00398
COMM SMOVL C00403 BC00403 V=1000.0  +MOVJ EC00399
COMM SFTOF3D
'EndPath W4844
'Path W4845
SFTOF3D
SFTON3D P028
MOVJ C00404 BC00404 VJ=100.00  +MOVJ EC00400 VJ=100.00
SMOVL C00405 BC00405 V=800.0  +MOVJ EC00401
SMOVL C00406 BC00406 V=150.0 PL=0  +MOVJ EC00402
MACRO1 MJ#(0) ARGF14
ARCON
SFTON3D P029
SMOVL C00407 BC00407 V=10.0  +MOVJ EC00403
SMOVL C00408 BC00408 V=10.0  +MOVJ EC00404
ARCOF
SMOVL C00409 BC00409 V=800.0  +MOVJ EC00405
SMOVL C00410 BC00410 V=1000.0  +MOVJ EC00406
SFTOF3D
'EndPath W4845
MOVJ C00411 BC00411 VJ=100.00  +MOVJ EC00407 VJ=100.00
MOVJ C00412 BC00412 VJ=100.00  +MOVJ EC00408 VJ=100.00
MOVJ C00413 BC00413 VJ=100.00  +MOVJ EC00409 VJ=100.00
'Path W4846
SFTOF3D
SFTON3D P030
MOVJ C00414 BC00414 VJ=100.00  +MOVJ EC00410 VJ=100.00
SMOVL C00415 BC00415 V=800.0  +MOVJ EC00411
SMOVL C00416 BC00416 V=150.0 PL=0  +MOVJ EC00412
ARCON
SMOVL C00417 BC00417 V=10.8  +MOVJ EC00413
SMOVL C00418 BC00418 V=10.8  +MOVJ EC00414
SMOVL C00419 BC00419 V=12.5  +MOVJ EC00415
SMOVL C00420 BC00420 V=12.5  +MOVJ EC00416
ARCOF
SMOVL C00421 BC00421 V=800.0  +MOVJ EC00417
SMOVL C00422 BC00422 V=1000.0  +MOVJ EC00418
SFTOF3D
'EndPath W4846
MOVJ C00423 BC00423 VJ=100.00  +MOVJ EC00419 VJ=100.00
MOVJ C00424 BC00424 VJ=100.00  +MOVJ EC00420 VJ=100.00
'Path W4847
SFTOF3D
SFTON3D P031
MOVJ C00425 BC00425 VJ=100.00  +MOVJ EC00421 VJ=100.00
SMOVL C00426 BC00426 V=800.0  +MOVJ EC00422
SMOVL C00427 BC00427 V=150.0 PL=0  +MOVJ EC00423
MACRO1 MJ#(0) ARGF9
ARCON
SWVON WEV#(101)
SMOVL C00428 BC00428 V=10.0 PL=0  +MOVJ EC00424
SMOVL C00429 BC00429 V=8.3  +MOVJ EC00425
SMOVL C00430 BC00430 V=8.3  +MOVJ EC00426
SWVOF
SFTON3D P030
SMOVL C00431 BC00431 V=10.0  +MOVJ EC00427
ARCOF
SMOVL C00432 BC00432 V=800.0  +MOVJ EC00428
SMOVL C00433 BC00433 V=1000.0  +MOVJ EC00429
SFTOF3D
'EndPath W4847
MOVJ C00434 BC00434 VJ=100.00  +MOVJ EC00430 VJ=100.00
MOVJ C00435 BC00435 VJ=100.00  +MOVJ EC00431 VJ=100.00
MACRO1 MJ#(0) ARGF6
MOVJ C00436 BC00436 VJ=100.00  +MOVJ EC00432 VJ=100.00
SFTON3D P045
SMOVL C00437 BC00437 V=133.3  +MOVJ EC00433
ARCON
SMOVL C00438 BC00438 V=11.7  +MOVJ EC00434
ARCOF
MOVJ C00439 BC00439 VJ=15.00  +MOVJ EC00435 VJ=100.00
MOVJ C00440 BC00440 VJ=80.00  +MOVJ EC00436 VJ=15.00
MOVJ C00441 BC00441 VJ=80.00  +MOVJ EC00437 VJ=80.00
SMOVL C00442 BC00442 V=133.3  +MOVJ EC00438
ARCON
SMOVL C00443 BC00443 V=11.7  +MOVJ EC00439
ARCOF
SMOVL C00444 BC00444 V=250.0  +MOVJ EC00440
SFTOF3D
MOVJ C00445 BC00445 VJ=80.00  +MOVJ EC00441 VJ=80.00
MOVJ C00446 BC00446 VJ=100.00  +MOVJ EC00442 VJ=100.00
END
